KUKA KRL program: EPS_2_25694_BP03_A_20251120043200.src

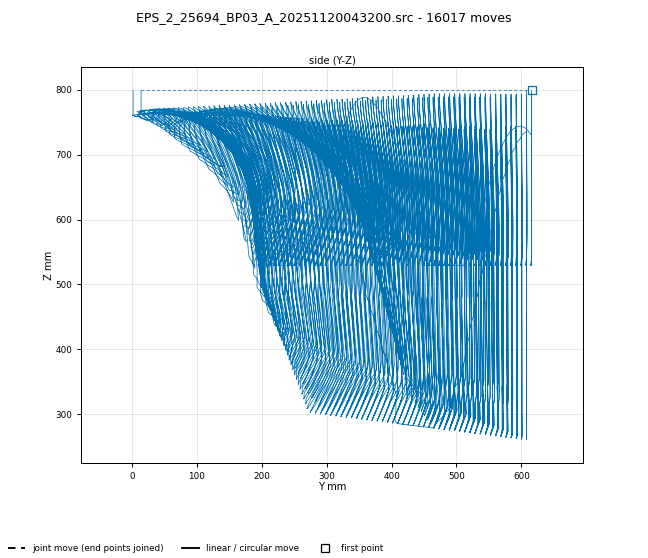
[picture p0: tool path of EPS_2_25694_BP03_A_20251120043200.src, 16017 of 16019 moves have a stored position in this frame; points joined in program order, loops and branches not executed]
&ACCESS RVP
&REL 4
&COMMENT QRS 19112012
&PARAM EDITMASK = *
DEF PART()
EXT BAS (BAS_COMMAND :IN,REAL :IN )
INT I
BAS (#INITMOV,0 )

;KUKA QRS Post kuka4.cps  Date:22-06-2017 !

File_ID=2926

QRS_PRE_INIT()

;Init var - Until changes are made in qrs_pre_init
Outlet_Square_prg=0
Inlet_1_Square_prg=0
Inlet_2_Square_prg=0
Inlet_3_Square_prg=0
Inlet_4_Square_prg=0
Inlet_5_Square_prg=0

Outlet_1={X 0.000, Y 466.000, Z 560.500, B 0.000, E1 0.000 }
Outlet_1={X 0.000, Y 466.000, Z 560.500, B 0.000, E1 0.000 }
Inlet_1={X 0.000, Y 466.000, Z 548.500, B 0.000, E1 90.000 }
Inlet_2={X 0.000, Y 519.840, Z 613.500, B 0.000, E1 205.000 }
Inlet_1={X 0.000, Y 466.000, Z 548.500, B 0.000, E1 90.000 }
Inlet_2={X 0.000, Y 519.840, Z 613.500, B 0.000, E1 205.000 }
Outlet_1_type=457
Inlet_1_type=381
Inlet_2_type=251
Inlet_1_type=381
Inlet_2_type=251
;QRS#1=Sidecore dimensions
;QRS#2=450-18" Concrete
;QRS#3=375-15" Concrete
;QRS#4=250-10" PVC SDR 35
;QRS#5=
;QRS#6=
;QRS#7=
;QRS#8=
;QRS#9=28A PSX-2
;QRS#10=24L PSX-2
;QRS#11=14M PSX
;QRS#12=
;QRS#13=
;QRS#14=
;QRS#15=
;QRS#16=1220x127x1143 3,75'
;QRS#17=EPS Height
;QRS#18=789
;QRS#19=*
;QRS#20= UPDATED VERSION 22-06-2017
;QRS#21=*
Outlet_Square=0250
Inlet_1_Square=0150
Inlet_2_Square=0100
Inlet_3_Square=0
Inlet_4_Square=0
Inlet_5_Square=0
Mill_Square=1
Outlet_Square_Prg=274
Inlet_1_Square_prg=261
Inlet_2_Square_prg=205
Inlet_1_Square_prg=261
Inlet_2_Square_prg=205

QRS_INIT()

$ADVANCE=5

; T1
PTP {E1 172.387,E2 172.387}
PTP {X 0,Y 615.713,A -85,B 0,C 180,E1 172.387,E2 172.387,E3 0,E4 0,E5 0,E6 0}
QRS_SPEED_INIT()
LIN {X 0,Y 615.713,Z 799,A -85,B 0,C 180,E1 172.387,E2 172.387,E3 0,E4 0,E5 0,E6 0} C_VEL
LIN {X 0,Y 615.713,Z 739.037,A -85,B 0,C 180,E1 172.387,E2 172.387} C_VEL
LIN {X 0,Y 615.713,Z 731.107,A -85,B 0,C 180,E1 172.387,E2 172.387} C_VEL
LIN {X 0,Y 615.691,Z 729.212,A -85,B 0,C 180,E1 172.633,E2 172.633} C_VEL
LIN {X 0,Y 615.732,Z 733.219,A -85,B 0,C 180,E1 173.736,E2 173.736} C_VEL
LIN {X 0,Y 615.814,Z 736.045,A -85,B 0,C 180,E1 174.659,E2 174.659} C_VEL
LIN {X 0,Y 615.663,Z 738.454,A -85,B 0,C 180,E1 175.589,E2 175.589} C_VEL
LIN {X 0,Y 615.667,Z 740.356,A -85,B 0,C 180,E1 176.519,E2 176.519} C_VEL
LIN {X 0,Y 615.819,Z 741.763,A -85,B 0,C 180,E1 177.448,E2 177.448} C_VEL
LIN {X 0,Y 615.624,Z 743.112,A -85,B 0,C 180,E1 178.84,E2 178.84} C_VEL
LIN {X 0,Y 615.601,Z 743.434,A -85,B 0,C 180,E1 179.768,E2 179.768} C_VEL
LIN {X 0,Y 615.739,Z 743.277,A -85,B 0,C 180,E1 180.696,E2 180.696} C_VEL
LIN {X 0,Y 615.854,Z 743.003,A -85,B 0,C 180,E1 181.159,E2 181.159} C_VEL
LIN {X 0,Y 615.71,Z 742.227,A -85,B 0,C 180,E1 182.088,E2 182.088} C_VEL
LIN {X 0,Y 615.687,Z 741.683,A -85,B 0,C 180,E1 182.552,E2 182.552} C_VEL
LIN {X 0,Y 615.745,Z 740.192,A -85,B 0,C 180,E1 183.481,E2 183.481} C_VEL
LIN {X 0,Y 615.79,Z 738.236,A -85,B 0,C 180,E1 184.41,E2 184.41} C_VEL
LIN {X 0,Y 615.65,Z 735.834,A -85,B 0,C 180,E1 185.342,E2 185.342} C_VEL
LIN {X 0,Y 615.661,Z 733.002,A -85,B 0,C 180,E1 186.247,E2 186.247} C_VEL
LIN {X 0,Y 615.81,Z 729.772,A -85,B 0,C 180,E1 187.122,E2 187.122} C_VEL
LIN {X 0,Y 615.717,Z 725.49,A -85,B 0,C 180,E1 188.145,E2 188.145} C_VEL
LIN {X 0,Y 615.668,Z 721.228,A -85,B 0,C 180,E1 189.025,E2 189.025} C_VEL
LIN {X 0,Y 615.787,Z 716.395,A -85,B 0,C 180,E1 189.905,E2 189.905} C_VEL
LIN {X 0,Y 615.78,Z 710.979,A -85,B 0,C 180,E1 190.789,E2 190.789} C_VEL
LIN {X 0,Y 615.717,Z 704.917,A -85,B 0,C 180,E1 191.677,E2 191.677} C_VEL
LIN {X 0,Y 615.775,Z 699.333,A -85,B 0,C 180,E1 192.417,E2 192.417} C_VEL
LIN {X 0,Y 615.828,Z 693.198,A -85,B 0,C 180,E1 193.158,E2 193.158} C_VEL
LIN {X 0,Y 615.758,Z 686.46,A -85,B 0,C 180,E1 193.905,E2 193.905} C_VEL
LIN {X 0,Y 615.758,Z 680.597,A -85,B 0,C 180,E1 194.503,E2 194.503} C_VEL
LIN {X 0,Y 615.803,Z 672.516,A -85,B 0,C 180,E1 195.252,E2 195.252} C_VEL
LIN {X 0,Y 615.785,Z 665.226,A -85,B 0,C 180,E1 195.871,E2 195.871} C_VEL
LIN {X 0,Y 615.783,Z 657.531,A -85,B 0,C 180,E1 196.468,E2 196.468} C_VEL
LIN {X 0,Y 615.772,Z 649.053,A -85,B 0,C 180,E1 197.069,E2 197.069} C_VEL
LIN {X 0,Y 615.777,Z 641.285,A -85,B 0,C 180,E1 197.571,E2 197.571} C_VEL
LIN {X 0,Y 615.791,Z 633.21,A -85,B 0,C 180,E1 198.046,E2 198.046} C_VEL
LIN {X 0,Y 615.786,Z 624.289,A -85,B 0,C 180,E1 198.521,E2 198.521} C_VEL
LIN {X 0,Y 615.708,Z 614.895,A -85,B 0,C 180,E1 198.971,E2 198.971} C_VEL
LIN {X 0,Y 615.796,Z 605.823,A -85,B 0,C 180,E1 199.352,E2 199.352} C_VEL
LIN {X 0,Y 615.802,Z 596.522,A -85,B 0,C 180,E1 199.698,E2 199.698} C_VEL
LIN {X 0,Y 615.75,Z 586.286,A -85,B 0,C 180,E1 200.027,E2 200.027} C_VEL
LIN {X 0,Y 615.701,Z 578.595,A -85,B 0,C 180,E1 200.243,E2 200.243} C_VEL
LIN {X 0,Y 615.799,Z 567.336,A -85,B 0,C 180,E1 200.495,E2 200.495} C_VEL
LIN {X 0,Y 615.798,Z 557.38,A -85,B 0,C 180,E1 200.672,E2 200.672} C_VEL
LIN {X 0,Y 615.482,Z 537.657,A -85,B 0,C 180,E1 200.94,E2 200.94} C_VEL
LIN {X 0,Y 615.266,Z 529.66,A -85,B 0,C 180,E1 201.046,E2 201.046} C_VEL
LIN {X 0,Y 615.471,Z 529.66,A -85,B 0,C 180,E1 201.079,E2 201.079} C_VEL
LIN {X 0,Y 615.868,Z 529.66,A -85,B 0,C 180,E1 201.381,E2 201.381} C_VEL
LIN {X 0,Y 615.844,Z 529.66,A -85,B 0,C 180,E1 202.61,E2 202.61} C_VEL
LIN {X 0,Y 615.752,Z 529.66,A -85,B 0,C 180,E1 207.74,E2 207.74} C_VEL
LIN {X 0,Y 615.186,Z 529.66,A -85,B 0,C 180,E1 210.425,E2 210.425} C_VEL
LIN {X 0,Y 615.704,Z 529.66,A -85,B 0,C 180,E1 213.124,E2 213.124} C_VEL
LIN {X 0,Y 615.633,Z 529.66,A -85,B 0,C 180,E1 213.911,E2 213.911} C_VEL
LIN {X 0,Y 615.66,Z 529.66,A -85,B 0,C 180,E1 218.863,E2 218.863} C_VEL
LIN {X 0,Y 615.247,Z 529.66,A -85,B 0,C 180,E1 221.943,E2 221.943} C_VEL
LIN {X 0,Y 615.648,Z 529.66,A -85,B 0,C 180,E1 224.892,E2 224.892} C_VEL
LIN {X 0,Y 615.652,Z 529.66,A -85,B 0,C 180,E1 228.496,E2 228.496} C_VEL
LIN {X 0,Y 615.387,Z 529.66,A -85,B 0,C 180,E1 231.116,E2 231.116} C_VEL
LIN {X 0,Y 615.438,Z 529.66,A -85,B 0,C 180,E1 232.155,E2 232.155} C_VEL
LIN {X 0,Y 615.703,Z 529.66,A -85,B 0,C 180,E1 234.059,E2 234.059} C_VEL
LIN {X 0,Y 615.162,Z 529.66,A -85,B 0,C 180,E1 236.842,E2 236.842} C_VEL
LIN {X 0,Y 615.753,Z 529.66,A -85,B 0,C 180,E1 239.606,E2 239.606} C_VEL
LIN {X 0,Y 615.248,Z 529.66,A -85,B 0,C 180,E1 242.234,E2 242.234} C_VEL
LIN {X 0,Y 615.196,Z 529.66,A -85,B 0,C 180,E1 244.825,E2 244.825} C_VEL
LIN {X 0,Y 614.949,Z 529.66,A -85,B 0,C 180,E1 244.857,E2 244.857} C_VEL
LIN {X 0,Y 615.521,Z 542.401,A -85,B 0,C 180,E1 245.055,E2 245.055} C_VEL
LIN {X 0,Y 615.592,Z 572.277,A -85,B 0,C 180,E1 245.446,E2 245.446} C_VEL
LIN {X 0,Y 615.552,Z 581.408,A -85,B 0,C 180,E1 245.594,E2 245.594} C_VEL
LIN {X 0,Y 615.691,Z 592.991,A -85,B 0,C 180,E1 245.841,E2 245.841} C_VEL
LIN {X 0,Y 615.671,Z 604.649,A -85,B 0,C 180,E1 246.141,E2 246.141} C_VEL
LIN {X 0,Y 615.619,Z 614.365,A -85,B 0,C 180,E1 246.431,E2 246.431} C_VEL
LIN {X 0,Y 615.762,Z 626.855,A -85,B 0,C 180,E1 246.881,E2 246.881} C_VEL
LIN {X 0,Y 615.772,Z 637.702,A -85,B 0,C 180,E1 247.323,E2 247.323} C_VEL
LIN {X 0,Y 615.696,Z 648.639,A -85,B 0,C 180,E1 247.826,E2 247.826} C_VEL
LIN {X 0,Y 615.747,Z 658.322,A -85,B 0,C 180,E1 248.324,E2 248.324} C_VEL
LIN {X 0,Y 615.764,Z 669.199,A -85,B 0,C 180,E1 248.948,E2 248.948} C_VEL
LIN {X 0,Y 615.755,Z 679.009,A -85,B 0,C 180,E1 249.567,E2 249.567} C_VEL
LIN {X 0,Y 615.75,Z 688.977,A -85,B 0,C 180,E1 250.261,E2 250.261} C_VEL
LIN {X 0,Y 615.756,Z 698.046,A -85,B 0,C 180,E1 250.953,E2 250.953} C_VEL
LIN {X 0,Y 615.778,Z 707.426,A -85,B 0,C 180,E1 251.737,E2 251.737} C_VEL
LIN {X 0,Y 615.74,Z 715.07,A -85,B 0,C 180,E1 252.428,E2 252.428} C_VEL
LIN {X 0,Y 615.695,Z 722.27,A -85,B 0,C 180,E1 253.13,E2 253.13} C_VEL
LIN {X 0,Y 615.739,Z 730.247,A -85,B 0,C 180,E1 253.981,E2 253.981} C_VEL
LIN {X 0,Y 615.804,Z 736.878,A -85,B 0,C 180,E1 254.747,E2 254.747} C_VEL
LIN {X 0,Y 615.686,Z 744.025,A -85,B 0,C 180,E1 255.644,E2 255.644} C_VEL
LIN {X 0,Y 615.686,Z 750.525,A -85,B 0,C 180,E1 256.54,E2 256.54} C_VEL
LIN {X 0,Y 615.815,Z 756.425,A -85,B 0,C 180,E1 257.435,E2 257.435} C_VEL
LIN {X 0,Y 615.707,Z 761.804,A -85,B 0,C 180,E1 258.322,E2 258.322} C_VEL
LIN {X 0,Y 615.618,Z 768.146,A -85,B 0,C 180,E1 259.503,E2 259.503} C_VEL
LIN {X 0,Y 615.746,Z 772.394,A -85,B 0,C 180,E1 260.388,E2 260.388} C_VEL
LIN {X 0,Y 615.772,Z 776.164,A -85,B 0,C 180,E1 261.269,E2 261.269} C_VEL
LIN {X 0,Y 615.627,Z 781.078,A -85,B 0,C 180,E1 262.578,E2 262.578} C_VEL
LIN {X 0,Y 615.759,Z 784.681,A -85,B 0,C 180,E1 263.749,E2 263.749} C_VEL
LIN {X 0,Y 615.831,Z 785.856,A -85,B 0,C 180,E1 264.192,E2 264.192} C_VEL
LIN {X 0,Y 615.723,Z 787.098,A -85,B 0,C 180,E1 264.657,E2 264.657} C_VEL
LIN {X 0,Y 615.589,Z 789.148,A -85,B 0,C 180,E1 265.587,E2 265.587} C_VEL
LIN {X 0,Y 615.603,Z 790.751,A -85,B 0,C 180,E1 266.518,E2 266.518} C_VEL
LIN {X 0,Y 615.787,Z 791.942,A -85,B 0,C 180,E1 267.447,E2 267.447} C_VEL
LIN {X 0,Y 615.603,Z 793.162,A -85,B 0,C 180,E1 268.839,E2 268.839} C_VEL
LIN {X 0,Y 615.579,Z 793.427,A -85,B 0,C 180,E1 269.767,E2 269.767} C_VEL
LIN {X 0,Y 615.832,Z 793.119,A -85,B 0,C 180,E1 271.158,E2 271.158} C_VEL
LIN {X 0,Y 615.72,Z 792.484,A -85,B 0,C 180,E1 272.087,E2 272.087} C_VEL
LIN {X 0,Y 615.801,Z 790.717,A -85,B 0,C 180,E1 273.479,E2 273.479} C_VEL
LIN {X 0,Y 615.711,Z 789.131,A -85,B 0,C 180,E1 274.41,E2 274.41} C_VEL
LIN {X 0,Y 615.574,Z 787.129,A -85,B 0,C 180,E1 275.342,E2 275.342} C_VEL
LIN {X 0,Y 615.634,Z 784.612,A -85,B 0,C 180,E1 276.287,E2 276.287} C_VEL
LIN {X 0,Y 615.792,Z 780.631,A -85,B 0,C 180,E1 277.55,E2 277.55} C_VEL
LIN {X 0,Y 615.625,Z 776.195,A -85,B 0,C 180,E1 278.731,E2 278.731} C_VEL
LIN {X 0,Y 615.66,Z 772.414,A -85,B 0,C 180,E1 279.611,E2 279.611} C_VEL
LIN {X 0,Y 615.799,Z 766.633,A -85,B 0,C 180,E1 280.787,E2 280.787} C_VEL
LIN {X 0,Y 615.638,Z 761.823,A -85,B 0,C 180,E1 281.677,E2 281.677} C_VEL
LIN {X 0,Y 615.663,Z 754.512,A -85,B 0,C 180,E1 282.863,E2 282.863} C_VEL
LIN {X 0,Y 615.826,Z 748.416,A -85,B 0,C 180,E1 283.753,E2 283.753} C_VEL
LIN {X 0,Y 615.735,Z 741.72,A -85,B 0,C 180,E1 284.653,E2 284.653} C_VEL
LIN {X 0,Y 615.701,Z 734.344,A -85,B 0,C 180,E1 285.553,E2 285.553} C_VEL
LIN {X 0,Y 615.778,Z 727.648,A -85,B 0,C 180,E1 286.305,E2 286.305} C_VEL
LIN {X 0,Y 615.765,Z 719.307,A -85,B 0,C 180,E1 287.163,E2 287.163} C_VEL
LIN {X 0,Y 615.713,Z 710.778,A -85,B 0,C 180,E1 287.968,E2 287.968} C_VEL
LIN {X 0,Y 615.737,Z 702.667,A -85,B 0,C 180,E1 288.671,E2 288.671} C_VEL
LIN {X 0,Y 615.745,Z 694.151,A -85,B 0,C 180,E1 289.352,E2 289.352} C_VEL
LIN {X 0,Y 615.759,Z 684.699,A -85,B 0,C 180,E1 290.045,E2 290.045} C_VEL
LIN {X 0,Y 615.742,Z 675.485,A -85,B 0,C 180,E1 290.663,E2 290.663} C_VEL
LIN {X 0,Y 615.716,Z 665.295,A -85,B 0,C 180,E1 291.285,E2 291.285} C_VEL
LIN {X 0,Y 615.75,Z 655.432,A -85,B 0,C 180,E1 291.83,E2 291.83} C_VEL
LIN {X 0,Y 615.747,Z 644.949,A -85,B 0,C 180,E1 292.352,E2 292.352} C_VEL
LIN {X 0,Y 615.698,Z 633.849,A -85,B 0,C 180,E1 292.844,E2 292.844} C_VEL
LIN {X 0,Y 615.669,Z 623.571,A -85,B 0,C 180,E1 293.249,E2 293.249} C_VEL
LIN {X 0,Y 615.734,Z 610.394,A -85,B 0,C 180,E1 293.687,E2 293.687} C_VEL
LIN {X 0,Y 615.669,Z 598.849,A -85,B 0,C 180,E1 294.016,E2 294.016} C_VEL
LIN {X 0,Y 615.62,Z 590.562,A -85,B 0,C 180,E1 294.221,E2 294.221} C_VEL
LIN {X 0,Y 615.768,Z 576.553,A -85,B 0,C 180,E1 294.483,E2 294.483} C_VEL
LIN {X 0,Y 615.688,Z 559.539,A -85,B 0,C 180,E1 294.722,E2 294.722} C_VEL
LIN {X 0,Y 615.448,Z 539.088,A -85,B 0,C 180,E1 294.99,E2 294.99} C_VEL
LIN {X 0,Y 614.945,Z 529.66,A -85,B 0,C 180,E1 295.141,E2 295.141} C_VEL
LIN {X 0,Y 615.189,Z 529.66,A -85,B 0,C 180,E1 295.173,E2 295.173} C_VEL
LIN {X 0,Y 615.248,Z 529.66,A -85,B 0,C 180,E1 297.764,E2 297.764} C_VEL
LIN {X 0,Y 615.753,Z 529.66,A -85,B 0,C 180,E1 300.392,E2 300.392} C_VEL
LIN {X 0,Y 615.154,Z 529.66,A -85,B 0,C 180,E1 303.845,E2 303.845} C_VEL
LIN {X 0,Y 615.702,Z 529.66,A -85,B 0,C 180,E1 305.938,E2 305.938} C_VEL
LIN {X 0,Y 615.768,Z 529.66,A -85,B 0,C 180,E1 308.853,E2 308.853} C_VEL
LIN {X 0,Y 615.261,Z 529.66,A -85,B 0,C 180,E1 311.94,E2 311.94} C_VEL
LIN {X 0,Y 615.681,Z 529.66,A -85,B 0,C 180,E1 314.895,E2 314.895} C_VEL
LIN {X 0,Y 615.647,Z 529.66,A -85,B 0,C 180,E1 318.495,E2 318.495} C_VEL
LIN {X 0,Y 615.364,Z 529.66,A -85,B 0,C 180,E1 321.115,E2 321.115} C_VEL
LIN {X 0,Y 615.416,Z 529.66,A -85,B 0,C 180,E1 322.155,E2 322.155} C_VEL
LIN {X 0,Y 615.67,Z 529.66,A -85,B 0,C 180,E1 324.058,E2 324.058} C_VEL
LIN {X 0,Y 615.141,Z 529.66,A -85,B 0,C 180,E1 326.841,E2 326.841} C_VEL
LIN {X 0,Y 615.744,Z 529.66,A -85,B 0,C 180,E1 329.606,E2 329.606} C_VEL
LIN {X 0,Y 615.231,Z 529.66,A -85,B 0,C 180,E1 332.234,E2 332.234} C_VEL
LIN {X 0,Y 615.765,Z 529.66,A -85,B 0,C 180,E1 334.851,E2 334.851} C_VEL
LIN {X 0,Y 615.775,Z 529.66,A -85,B 0,C 180,E1 339.878,E2 339.878} C_VEL
LIN {X 0,Y 615.792,Z 529.66,A -85,B 0,C 180,E1 343.784,E2 343.784} C_VEL
LIN {X 0,Y 615.824,Z 529.66,A -85,B 0,C 180,E1 349.507,E2 349.507} C_VEL
LIN {X 0,Y 615.819,Z 529.66,A -85,B 0,C 180,E1 354.193,E2 354.193} C_VEL
LIN {X 0,Y 615.867,Z 529.66,A -85,B 0,C 180,E1 358.841,E2 358.841} C_VEL
LIN {X 0,Y 615.87,Z 529.66,A -85,B 0,C 180,E1 363.48,E2 363.48} C_VEL
LIN {X 0,Y 615.807,Z 529.66,A -85,B 0,C 180,E1 368.143,E2 368.143} C_VEL
LIN {X 0,Y 615.817,Z 529.66,A -85,B 0,C 180,E1 372.861,E2 372.861} C_VEL
LIN {X 0,Y 615.8,Z 529.66,A -85,B 0,C 180,E1 377.67,E2 377.67} C_VEL
LIN {X 0,Y 615.799,Z 529.66,A -85,B 0,C 180,E1 377.998,E2 377.998} C_VEL
LIN {X 0,Y 615.759,Z 529.66,A -85,B 0,C 180,E1 382.613,E2 382.613} C_VEL
LIN {X 0,Y 615.223,Z 529.66,A -85,B 0,C 180,E1 385.173,E2 385.173} C_VEL
LIN {X 0,Y 615.722,Z 529.66,A -85,B 0,C 180,E1 387.742,E2 387.742} C_VEL
LIN {X 0,Y 615.171,Z 529.66,A -85,B 0,C 180,E1 390.426,E2 390.426} C_VEL
LIN {X 0,Y 615.705,Z 529.66,A -85,B 0,C 180,E1 393.124,E2 393.124} C_VEL
LIN {X 0,Y 615.647,Z 529.66,A -85,B 0,C 180,E1 393.916,E2 393.916} C_VEL
LIN {X 0,Y 615.662,Z 529.66,A -85,B 0,C 180,E1 398.863,E2 398.863} C_VEL
LIN {X 0,Y 615.226,Z 529.66,A -85,B 0,C 180,E1 401.945,E2 401.945} C_VEL
LIN {X 0,Y 615.622,Z 529.66,A -85,B 0,C 180,E1 404.892,E2 404.892} C_VEL
LIN {X 0,Y 615.63,Z 529.66,A -85,B 0,C 180,E1 408.499,E2 408.499} C_VEL
LIN {X 0,Y 615.634,Z 529.66,A -85,B 0,C 180,E1 409.224,E2 409.224} C_VEL
LIN {X 0,Y 614.905,Z 529.66,A -85,B 0,C 180,E1 409.372,E2 409.372} C_VEL
LIN {X 0,Y 614.377,Z 529.66,A -85,B 0,C 180,E1 409.433,E2 409.433} C_VEL
LIN {X 0,Y 614.179,Z 530.164,A -85,B 0,C 180,E1 409.484,E2 409.484} C_VEL
LIN {X 0,Y 615.256,Z 532.913,A -85,B 0,C 180,E1 409.545,E2 409.545} C_VEL
LIN {X 0,Y 615.716,Z 535.143,A -85,B 0,C 180,E1 409.583,E2 409.583} C_VEL
LIN {X 0,Y 615.768,Z 609.489,A -85,B 0,C 180,E1 410.467,E2 410.467} C_VEL
LIN {X 0,Y 615.796,Z 617.276,A -85,B 0,C 180,E1 410.59,E2 410.59} C_VEL
LIN {X 0,Y 615.762,Z 625.824,A -85,B 0,C 180,E1 410.767,E2 410.767} C_VEL
LIN {X 0,Y 615.8,Z 635.584,A -85,B 0,C 180,E1 411.03,E2 411.03} C_VEL
LIN {X 0,Y 615.784,Z 644.692,A -85,B 0,C 180,E1 411.34,E2 411.34} C_VEL
LIN {X 0,Y 615.833,Z 653.267,A -85,B 0,C 180,E1 411.687,E2 411.687} C_VEL
LIN {X 0,Y 615.837,Z 663.366,A -85,B 0,C 180,E1 412.173,E2 412.173} C_VEL
LIN {X 0,Y 615.838,Z 670.383,A -85,B 0,C 180,E1 412.565,E2 412.565} C_VEL
LIN {X 0,Y 615.802,Z 678.254,A -85,B 0,C 180,E1 413.06,E2 413.06} C_VEL
LIN {X 0,Y 615.823,Z 685.634,A -85,B 0,C 180,E1 413.59,E2 413.59} C_VEL
LIN {X 0,Y 615.832,Z 693.033,A -85,B 0,C 180,E1 414.194,E2 414.194} C_VEL
LIN {X 0,Y 615.776,Z 699.754,A -85,B 0,C 180,E1 414.807,E2 414.807} C_VEL
LIN {X 0,Y 615.778,Z 705.651,A -85,B 0,C 180,E1 415.419,E2 415.419} C_VEL
LIN {X 0,Y 615.83,Z 711.178,A -85,B 0,C 180,E1 416.062,E2 416.062} C_VEL
LIN {X 0,Y 615.759,Z 717.457,A -85,B 0,C 180,E1 416.881,E2 416.881} C_VEL
LIN {X 0,Y 615.743,Z 722.895,A -85,B 0,C 180,E1 417.715,E2 417.715} C_VEL
LIN {X 0,Y 615.829,Z 726.982,A -85,B 0,C 180,E1 418.434,E2 418.434} C_VEL
LIN {X 0,Y 615.789,Z 730.525,A -85,B 0,C 180,E1 419.14,E2 419.14} C_VEL
LIN {X 0,Y 615.712,Z 734.28,A -85,B 0,C 180,E1 420.032,E2 420.032} C_VEL
LIN {X 0,Y 615.725,Z 735.961,A -85,B 0,C 180,E1 420.488,E2 420.488} C_VEL
LIN {X 0,Y 615.843,Z 738.595,A -85,B 0,C 180,E1 421.365,E2 421.365} C_VEL
LIN {X 0,Y 615.741,Z 740.746,A -85,B 0,C 180,E1 422.261,E2 422.261} C_VEL
LIN {X 0,Y 615.727,Z 741.895,A -85,B 0,C 180,E1 422.913,E2 422.913} C_VEL
LIN {X 0,Y 615.792,Z 742.709,A -85,B 0,C 180,E1 423.565,E2 423.565} C_VEL
LIN {X 0,Y 615.815,Z 743.213,A -85,B 0,C 180,E1 424.212,E2 424.212} C_VEL
LIN {X 0,Y 615.733,Z 743.429,A -85,B 0,C 180,E1 424.851,E2 424.851} C_VEL
LIN {X 0,Y 615.737,Z 743.29,A -85,B 0,C 180,E1 425.605,E2 425.605} C_VEL
LIN {X 0,Y 615.851,Z 742.529,A -85,B 0,C 180,E1 426.486,E2 426.486} C_VEL
LIN {X 0,Y 615.727,Z 741.246,A -85,B 0,C 180,E1 427.387,E2 427.387} C_VEL
LIN {X 0,Y 615.686,Z 739.971,A -85,B 0,C 180,E1 428.012,E2 428.012} C_VEL
LIN {X 0,Y 615.727,Z 738.372,A -85,B 0,C 180,E1 428.637,E2 428.637} C_VEL
LIN {X 0,Y 615.814,Z 735.406,A -85,B 0,C 180,E1 429.571,E2 429.571} C_VEL
LIN {X 0,Y 615.73,Z 731.754,A -85,B 0,C 180,E1 430.494,E2 430.494} C_VEL
LIN {X 0,Y 615.777,Z 727.849,A -85,B 0,C 180,E1 431.318,E2 431.318} C_VEL
LIN {X 0,Y 615.82,Z 723.223,A -85,B 0,C 180,E1 432.138,E2 432.138} C_VEL
LIN {X 0,Y 615.771,Z 719.45,A -85,B 0,C 180,E1 432.734,E2 432.734} C_VEL
LIN {X 0,Y 615.775,Z 715.176,A -85,B 0,C 180,E1 433.338,E2 433.338} C_VEL
LIN {X 0,Y 615.841,Z 708.758,A -85,B 0,C 180,E1 434.141,E2 434.141} C_VEL
LIN {X 0,Y 615.801,Z 703.223,A -85,B 0,C 180,E1 434.749,E2 434.749} C_VEL
LIN {X 0,Y 615.796,Z 697.131,A -85,B 0,C 180,E1 435.349,E2 435.349} C_VEL
LIN {X 0,Y 615.844,Z 690.323,A -85,B 0,C 180,E1 435.948,E2 435.948} C_VEL
LIN {X 0,Y 615.841,Z 682.573,A -85,B 0,C 180,E1 436.545,E2 436.545} C_VEL
LIN {X 0,Y 615.837,Z 674.946,A -85,B 0,C 180,E1 437.066,E2 437.066} C_VEL
LIN {X 0,Y 615.813,Z 666.212,A -85,B 0,C 180,E1 437.585,E2 437.585} C_VEL
LIN {X 0,Y 615.845,Z 657.471,A -85,B 0,C 180,E1 438.031,E2 438.031} C_VEL
LIN {X 0,Y 615.83,Z 649.113,A -85,B 0,C 180,E1 438.401,E2 438.401} C_VEL
LIN {X 0,Y 615.771,Z 640.154,A -85,B 0,C 180,E1 438.732,E2 438.732} C_VEL
LIN {X 0,Y 615.831,Z 630.951,A -85,B 0,C 180,E1 439.01,E2 439.01} C_VEL
LIN {X 0,Y 615.801,Z 621.089,A -85,B 0,C 180,E1 439.25,E2 439.25} C_VEL
LIN {X 0,Y 615.781,Z 611.462,A -85,B 0,C 180,E1 439.415,E2 439.415} C_VEL
LIN {X 0,Y 615.609,Z 555.605,A -85,B 0,C 180,E1 440.088,E2 440.088} C_VEL
LIN {X 0,Y 615.309,Z 530.18,A -85,B 0,C 180,E1 440.396,E2 440.396} C_VEL
LIN {X 0,Y 615.401,Z 529.66,A -85,B 0,C 180,E1 440.42,E2 440.42} C_VEL
LIN {X 0,Y 615.834,Z 529.66,A -85,B 0,C 180,E1 440.539,E2 440.539} C_VEL
LIN {X 0,Y 615.861,Z 529.66,A -85,B 0,C 180,E1 446.521,E2 446.521} C_VEL
LIN {X 0,Y 615.873,Z 529.66,A -85,B 0,C 180,E1 451.16,E2 451.16} C_VEL
LIN {X 0,Y 615.873,Z 529.66,A -85,B 0,C 180,E1 455.807,E2 455.807} C_VEL
LIN {X 0,Y 615.788,Z 529.66,A -85,B 0,C 180,E1 460.495,E2 460.495} C_VEL
LIN {X 0,Y 615.769,Z 529.66,A -85,B 0,C 180,E1 465.254,E2 465.254} C_VEL
LIN {X 0,Y 615.782,Z 529.66,A -85,B 0,C 180,E1 470.123,E2 470.123} C_VEL
LIN {X 0,Y 615.745,Z 529.66,A -85,B 0,C 180,E1 475.151,E2 475.151} C_VEL
LIN {X 0,Y 615.396,Z 529.66,A -85,B 0,C 180,E1 479.457,E2 479.457} C_VEL
LIN {X 0,Y 615.719,Z 529.66,A -85,B 0,C 180,E1 480.396,E2 480.396} C_VEL
LIN {X 0,Y 615.15,Z 529.66,A -85,B 0,C 180,E1 483.844,E2 483.844} C_VEL
LIN {X 0,Y 615.698,Z 529.66,A -85,B 0,C 180,E1 485.941,E2 485.941} C_VEL
LIN {X 0,Y 615.668,Z 529.66,A -85,B 0,C 180,E1 487.873,E2 487.873} C_VEL
LIN {X 0,Y 615.757,Z 529.66,A -85,B 0,C 180,E1 488.856,E2 488.856} C_VEL
LIN {X 0,Y 615.253,Z 529.66,A -85,B 0,C 180,E1 491.943,E2 491.943} C_VEL
LIN {X 0,Y 615.673,Z 529.66,A -85,B 0,C 180,E1 494.894,E2 494.894} C_VEL
LIN {X 0,Y 615.655,Z 529.66,A -85,B 0,C 180,E1 498.497,E2 498.497} C_VEL
LIN {X 0,Y 615.36,Z 529.66,A -85,B 0,C 180,E1 501.114,E2 501.114} C_VEL
LIN {X 0,Y 615.396,Z 529.66,A -85,B 0,C 180,E1 502.16,E2 502.16} C_VEL
LIN {X 0,Y 615.651,Z 529.66,A -85,B 0,C 180,E1 504.056,E2 504.056} C_VEL
LIN {X 0,Y 615.118,Z 529.66,A -85,B 0,C 180,E1 506.84,E2 506.84} C_VEL
LIN {X 0,Y 615.715,Z 529.66,A -85,B 0,C 180,E1 509.604,E2 509.604} C_VEL
LIN {X 0,Y 615.228,Z 529.66,A -85,B 0,C 180,E1 512.234,E2 512.234} C_VEL
LIN {X 0,Y 615.796,Z 529.66,A -85,B 0,C 180,E1 514.852,E2 514.852} C_VEL
LIN {X 0,Y 615.831,Z 529.66,A -85,B 0,C 180,E1 518.764,E2 518.764} C_VEL
LIN {X 0,Y 615.602,Z 529.66,A -85,B 0,C 180,E1 518.876,E2 518.876} C_VEL
LIN {X 0,Y 615.779,Z 556.304,A -85,B 0,C 180,E1 519.221,E2 519.221} C_VEL
LIN {X 0,Y 615.741,Z 565.587,A -85,B 0,C 180,E1 519.379,E2 519.379} C_VEL
LIN {X 0,Y 615.667,Z 573.153,A -85,B 0,C 180,E1 519.536,E2 519.536} C_VEL
LIN {X 0,Y 615.78,Z 583.294,A -85,B 0,C 180,E1 519.798,E2 519.798} C_VEL
LIN {X 0,Y 615.784,Z 592.324,A -85,B 0,C 180,E1 520.071,E2 520.071} C_VEL
LIN {X 0,Y 615.688,Z 602.19,A -85,B 0,C 180,E1 520.414,E2 520.414} C_VEL
LIN {X 0,Y 615.79,Z 611.709,A -85,B 0,C 180,E1 520.802,E2 520.802} C_VEL
LIN {X 0,Y 615.797,Z 620.728,A -85,B 0,C 180,E1 521.213,E2 521.213} C_VEL
LIN {X 0,Y 615.785,Z 628.975,A -85,B 0,C 180,E1 521.631,E2 521.631} C_VEL
LIN {X 0,Y 615.757,Z 637.944,A -85,B 0,C 180,E1 522.136,E2 522.136} C_VEL
LIN {X 0,Y 615.78,Z 645.951,A -85,B 0,C 180,E1 522.633,E2 522.633} C_VEL
LIN {X 0,Y 615.797,Z 654.793,A -85,B 0,C 180,E1 523.241,E2 523.241} C_VEL
LIN {X 0,Y 615.791,Z 662.806,A -85,B 0,C 180,E1 523.845,E2 523.845} C_VEL
LIN {X 0,Y 615.765,Z 670.118,A -85,B 0,C 180,E1 524.447,E2 524.447} C_VEL
LIN {X 0,Y 615.769,Z 676.821,A -85,B 0,C 180,E1 525.047,E2 525.047} C_VEL
LIN {X 0,Y 615.814,Z 683.003,A -85,B 0,C 180,E1 525.648,E2 525.648} C_VEL
LIN {X 0,Y 615.765,Z 690.046,A -85,B 0,C 180,E1 526.393,E2 526.393} C_VEL
LIN {X 0,Y 615.709,Z 696.458,A -85,B 0,C 180,E1 527.136,E2 527.136} C_VEL
LIN {X 0,Y 615.756,Z 702.296,A -85,B 0,C 180,E1 527.88,E2 527.88} C_VEL
LIN {X 0,Y 615.831,Z 707.614,A -85,B 0,C 180,E1 528.621,E2 528.621} C_VEL
LIN {X 0,Y 615.73,Z 711.581,A -85,B 0,C 180,E1 529.21,E2 529.21} C_VEL
LIN {X 0,Y 615.661,Z 716.922,A -85,B 0,C 180,E1 530.093,E2 530.093} C_VEL
LIN {X 0,Y 615.762,Z 721.658,A -85,B 0,C 180,E1 530.977,E2 530.977} C_VEL
LIN {X 0,Y 615.79,Z 725.868,A -85,B 0,C 180,E1 531.856,E2 531.856} C_VEL
LIN {X 0,Y 615.691,Z 729.212,A -85,B 0,C 180,E1 532.633,E2 532.633} C_VEL
LIN {X 0,Y 611.74,Z 735.059,A -85,B 0,C 180,E1 534.144,E2 534.144} C_VEL
LIN {X 0,Y 607.783,Z 739.278,A -85,B 0,C 180,E1 535.697,E2 535.697} C_VEL
LIN {X 0,Y 607.763,Z 743.464,A -85,B 0,C 180,E1 538.575,E2 538.575} C_VEL
LIN {X 0,Y 607.922,Z 743.404,A -85,B 0,C 180,E1 541.42,E2 541.42} C_VEL
LIN {X 0,Y 607.899,Z 739.162,A -85,B 0,C 180,E1 544.269,E2 544.269} C_VEL
LIN {X 0,Y 607.883,Z 728.493,A -85,B 0,C 180,E1 547.623,E2 547.623} C_VEL
LIN {X 0,Y 607.939,Z 712.456,A -85,B 0,C 180,E1 550.727,E2 550.727} C_VEL
LIN {X 0,Y 608,Z 692.204,A -85,B 0,C 180,E1 553.453,E2 553.453} C_VEL
LIN {X 0,Y 608.082,Z 667.028,A -85,B 0,C 180,E1 555.931,E2 555.931} C_VEL
LIN {X 0,Y 608.185,Z 638.464,A -85,B 0,C 180,E1 557.972,E2 557.972} C_VEL
LIN {X 0,Y 608.294,Z 606.206,A -85,B 0,C 180,E1 559.586,E2 559.586} C_VEL
LIN {X 0,Y 608.364,Z 572.382,A -85,B 0,C 180,E1 560.649,E2 560.649} C_VEL
LIN {X 0,Y 607.906,Z 529.66,A -85,B 0,C 180,E1 561.38,E2 561.38} C_VEL
LIN {X 0,Y 607.695,Z 529.66,A -85,B 0,C 180,E1 568.148,E2 568.148} C_VEL
LIN {X 0,Y 607.809,Z 529.66,A -85,B 0,C 180,E1 573.103,E2 573.103} C_VEL
LIN {X 0,Y 607.507,Z 529.66,A -85,B 0,C 180,E1 579.646,E2 579.646} C_VEL
LIN {X 0,Y 607.506,Z 529.66,A -85,B 0,C 180,E1 585.934,E2 585.934} C_VEL
LIN {X 0,Y 607.452,Z 529.66,A -85,B 0,C 180,E1 590.357,E2 590.357} C_VEL
LIN {X 0,Y 607.433,Z 529.66,A -85,B 0,C 180,E1 595.155,E2 595.155} C_VEL
LIN {X 0,Y 607.601,Z 529.66,A -85,B 0,C 180,E1 600.365,E2 600.365} C_VEL
LIN {X 0,Y 607.26,Z 529.66,A -85,B 0,C 180,E1 604.503,E2 604.503} C_VEL
LIN {X 0,Y 608.436,Z 561.303,A -85,B 0,C 180,E1 604.986,E2 604.986} C_VEL
LIN {X 0,Y 608.473,Z 599.633,A -85,B 0,C 180,E1 605.701,E2 605.701} C_VEL
LIN {X 0,Y 608.446,Z 636.055,A -85,B 0,C 180,E1 606.96,E2 606.96} C_VEL
LIN {X 0,Y 608.25,Z 670.026,A -85,B 0,C 180,E1 608.727,E2 608.727} C_VEL
LIN {X 0,Y 608.111,Z 700.158,A -85,B 0,C 180,E1 610.879,E2 610.879} C_VEL
LIN {X 0,Y 607.968,Z 728.788,A -85,B 0,C 180,E1 613.601,E2 613.601} C_VEL
LIN {X 0,Y 607.882,Z 751.803,A -85,B 0,C 180,E1 616.543,E2 616.543} C_VEL
LIN {X 0,Y 607.8,Z 769.647,A -85,B 0,C 180,E1 619.631,E2 619.631} C_VEL
LIN {X 0,Y 607.768,Z 782.683,A -85,B 0,C 180,E1 622.869,E2 622.869} C_VEL
LIN {X 0,Y 607.71,Z 789.996,A -85,B 0,C 180,E1 625.729,E2 625.729} C_VEL
LIN {X 0,Y 607.739,Z 793.511,A -85,B 0,C 180,E1 628.578,E2 628.578} C_VEL
LIN {X 0,Y 607.908,Z 793.51,A -85,B 0,C 180,E1 631.423,E2 631.423} C_VEL
LIN {X 0,Y 607.73,Z 788.487,A -85,B 0,C 180,E1 634.986,E2 634.986} C_VEL
LIN {X 0,Y 607.83,Z 778.937,A -85,B 0,C 180,E1 638.208,E2 638.208} C_VEL
LIN {X 0,Y 607.838,Z 764.016,A -85,B 0,C 180,E1 641.456,E2 641.456} C_VEL
LIN {X 0,Y 607.963,Z 744.066,A -85,B 0,C 180,E1 644.545,E2 644.545} C_VEL
LIN {X 0,Y 608.05,Z 718.03,A -85,B 0,C 180,E1 647.513,E2 647.513} C_VEL
LIN {X 0,Y 608.194,Z 688.345,A -85,B 0,C 180,E1 650.042,E2 650.042} C_VEL
LIN {X 0,Y 608.316,Z 654.998,A -85,B 0,C 180,E1 652.133,E2 652.133} C_VEL
LIN {X 0,Y 608.392,Z 620.469,A -85,B 0,C 180,E1 653.653,E2 653.653} C_VEL
LIN {X 0,Y 608.477,Z 586.214,A -85,B 0,C 180,E1 654.613,E2 654.613} C_VEL
LIN {X 0,Y 607.58,Z 531.954,A -85,B 0,C 180,E1 655.428,E2 655.428} C_VEL
LIN {X 0,Y 607.239,Z 529.66,A -85,B 0,C 180,E1 655.538,E2 655.538} C_VEL
LIN {X 0,Y 607.647,Z 529.66,A -85,B 0,C 180,E1 659.78,E2 659.78} C_VEL
LIN {X 0,Y 607.71,Z 529.66,A -85,B 0,C 180,E1 666.58,E2 666.58} C_VEL
LIN {X 0,Y 607.339,Z 529.66,A -85,B 0,C 180,E1 672.133,E2 672.133} C_VEL
LIN {X 0,Y 607.666,Z 529.66,A -85,B 0,C 180,E1 678.158,E2 678.158} C_VEL
LIN {X 0,Y 607.629,Z 529.66,A -85,B 0,C 180,E1 683.418,E2 683.418} C_VEL
LIN {X 0,Y 607.566,Z 529.66,A -85,B 0,C 180,E1 690.377,E2 690.377} C_VEL
LIN {X 0,Y 607.799,Z 529.66,A -85,B 0,C 180,E1 695.038,E2 695.038} C_VEL
LIN {X 0,Y 607.569,Z 529.66,A -85,B 0,C 180,E1 701.165,E2 701.165} C_VEL
LIN {X 0,Y 607.264,Z 529.66,A -85,B 0,C 180,E1 705.614,E2 705.614} C_VEL
LIN {X 0,Y 607.746,Z 529.66,A -85,B 0,C 180,E1 709.993,E2 709.993} C_VEL
LIN {X 0,Y 607.881,Z 529.66,A -85,B 0,C 180,E1 714.303,E2 714.303} C_VEL
LIN {X 0,Y 607.588,Z 529.66,A -85,B 0,C 180,E1 720.002,E2 720.002} C_VEL
LIN {X 0,Y 607.67,Z 529.66,A -85,B 0,C 180,E1 724.274,E2 724.274} C_VEL
LIN {X 0,Y 607.764,Z 529.66,A -85,B 0,C 180,E1 728.569,E2 728.569} C_VEL
LIN {X 0,Y 607.888,Z 529.66,A -85,B 0,C 180,E1 732.911,E2 732.911} C_VEL
LIN {X 0,Y 607.594,Z 529.66,A -85,B 0,C 180,E1 738.838,E2 738.838} C_VEL
LIN {X 0,Y 607.579,Z 529.66,A -85,B 0,C 180,E1 743.416,E2 743.416} C_VEL
LIN {X 0,Y 607.658,Z 529.66,A -85,B 0,C 180,E1 748.155,E2 748.155} C_VEL
LIN {X 0,Y 607.808,Z 529.66,A -85,B 0,C 180,E1 753.108,E2 753.108} C_VEL
LIN {X 0,Y 607.482,Z 529.66,A -85,B 0,C 180,E1 759.641,E2 759.641} C_VEL
LIN {X 0,Y 607.495,Z 529.66,A -85,B 0,C 180,E1 765.931,E2 765.931} C_VEL
LIN {X 0,Y 607.177,Z 529.66,A -85,B 0,C 180,E1 769.131,E2 769.131} C_VEL
LIN {X 0,Y 606.592,Z 530.446,A -85,B 0,C 180,E1 769.289,E2 769.289} C_VEL
LIN {X 0,Y 608.098,Z 542.16,A -85,B 0,C 180,E1 769.47,E2 769.47} C_VEL
LIN {X 0,Y 608.144,Z 624.143,A -85,B 0,C 180,E1 770.546,E2 770.546} C_VEL
LIN {X 0,Y 608.124,Z 652.634,A -85,B 0,C 180,E1 771.488,E2 771.488} C_VEL
LIN {X 0,Y 608.039,Z 678.51,A -85,B 0,C 180,E1 772.92,E2 772.92} C_VEL
LIN {X 0,Y 607.96,Z 701.929,A -85,B 0,C 180,E1 774.882,E2 774.882} C_VEL
LIN {X 0,Y 607.914,Z 721.026,A -85,B 0,C 180,E1 777.267,E2 777.267} C_VEL
LIN {X 0,Y 607.858,Z 734.168,A -85,B 0,C 180,E1 779.82,E2 779.82} C_VEL
LIN {X 0,Y 607.917,Z 740.473,A -85,B 0,C 180,E1 781.86,E2 781.86} C_VEL
LIN {X 0,Y 607.925,Z 743.162,A -85,B 0,C 180,E1 783.461,E2 783.461} C_VEL
LIN {X 0,Y 607.861,Z 743.988,A -85,B 0,C 180,E1 785.037,E2 785.037} C_VEL
LIN {X 0,Y 607.866,Z 741.852,A -85,B 0,C 180,E1 787.369,E2 787.369} C_VEL
LIN {X 0,Y 607.924,Z 734.675,A -85,B 0,C 180,E1 789.953,E2 789.953} C_VEL
LIN {X 0,Y 607.958,Z 722.026,A -85,B 0,C 180,E1 792.485,E2 792.485} C_VEL
LIN {X 0,Y 607.989,Z 704.616,A -85,B 0,C 180,E1 794.749,E2 794.749} C_VEL
LIN {X 0,Y 608.055,Z 682.187,A -85,B 0,C 180,E1 796.729,E2 796.729} C_VEL
LIN {X 0,Y 608.143,Z 655.872,A -85,B 0,C 180,E1 798.278,E2 798.278} C_VEL
LIN {X 0,Y 608.174,Z 627.894,A -85,B 0,C 180,E1 799.275,E2 799.275} C_VEL
LIN {X 0,Y 608.067,Z 586.852,A -85,B 0,C 180,E1 799.905,E2 799.905} C_VEL
LIN {X 0,Y 607.797,Z 529.66,A -85,B 0,C 180,E1 800.612,E2 800.612} C_VEL
LIN {X 0,Y 607.737,Z 529.66,A -85,B 0,C 180,E1 807.153,E2 807.153} C_VEL
LIN {X 0,Y 607.866,Z 529.66,A -85,B 0,C 180,E1 811.422,E2 811.422} C_VEL
LIN {X 0,Y 607.663,Z 529.66,A -85,B 0,C 180,E1 816.622,E2 816.622} C_VEL
LIN {X 0,Y 607.559,Z 529.66,A -85,B 0,C 180,E1 821.46,E2 821.46} C_VEL
LIN {X 0,Y 607.629,Z 529.66,A -85,B 0,C 180,E1 825.853,E2 825.853} C_VEL
LIN {X 0,Y 607.785,Z 529.66,A -85,B 0,C 180,E1 830.339,E2 830.339} C_VEL
LIN {X 0,Y 607.782,Z 529.66,A -85,B 0,C 180,E1 834.965,E2 834.965} C_VEL
LIN {X 0,Y 607.605,Z 529.66,A -85,B 0,C 180,E1 839.781,E2 839.781} C_VEL
LIN {X 0,Y 607.731,Z 529.66,A -85,B 0,C 180,E1 846.577,E2 846.577} C_VEL
LIN {X 0,Y 607.338,Z 529.66,A -85,B 0,C 180,E1 851.806,E2 851.806} C_VEL
LIN {X 0,Y 607.499,Z 529.66,A -85,B 0,C 180,E1 856.082,E2 856.082} C_VEL
LIN {X 0,Y 607.414,Z 529.66,A -85,B 0,C 180,E1 860.364,E2 860.364} C_VEL
LIN {X 0,Y 607.386,Z 529.66,A -85,B 0,C 180,E1 865.149,E2 865.149} C_VEL
LIN {X 0,Y 607.554,Z 529.66,A -85,B 0,C 180,E1 870.376,E2 870.376} C_VEL
LIN {X 0,Y 607.839,Z 529.66,A -85,B 0,C 180,E1 875.035,E2 875.035} C_VEL
LIN {X 0,Y 607.876,Z 529.66,A -85,B 0,C 180,E1 878.591,E2 878.591} C_VEL
LIN {X 0,Y 608.277,Z 575.93,A -85,B 0,C 180,E1 879.344,E2 879.344} C_VEL
LIN {X 0,Y 608.263,Z 610.705,A -85,B 0,C 180,E1 880.51,E2 880.51} C_VEL
LIN {X 0,Y 608.17,Z 642.889,A -85,B 0,C 180,E1 882.21,E2 882.21} C_VEL
LIN {X 0,Y 608.047,Z 672.15,A -85,B 0,C 180,E1 884.425,E2 884.425} C_VEL
LIN {X 0,Y 607.904,Z 697.501,A -85,B 0,C 180,E1 887.089,E2 887.089} C_VEL
LIN {X 0,Y 607.809,Z 717.287,A -85,B 0,C 180,E1 889.99,E2 889.99} C_VEL
LIN {X 0,Y 607.812,Z 730.807,A -85,B 0,C 180,E1 892.867,E2 892.867} C_VEL
LIN {X 0,Y 607.783,Z 739.278,A -85,B 0,C 180,E1 895.697,E2 895.697} C_VEL
LIN {X 0,Y 605.253,Z 741.666,A -85,B 0,C 180,E1 896.89,E2 896.89} C_VEL
LIN {X 0,Y 599.93,Z 743.564,A -85,B 0,C 180,E1 898.698,E2 898.698} C_VEL
LIN {X 0,Y 599.824,Z 743.595,A -85,B 0,C 180,E1 898.908,E2 898.908} C_VEL
LIN {X 0,Y 600.018,Z 743.406,A -85,B 0,C 180,E1 901.439,E2 901.439} C_VEL
LIN {X 0,Y 600.013,Z 739.166,A -85,B 0,C 180,E1 904.325,E2 904.325} C_VEL
LIN {X 0,Y 599.998,Z 729.078,A -85,B 0,C 180,E1 907.585,E2 907.585} C_VEL
LIN {X 0,Y 600.078,Z 713.416,A -85,B 0,C 180,E1 910.708,E2 910.708} C_VEL
LIN {X 0,Y 600.21,Z 692.212,A -85,B 0,C 180,E1 913.631,E2 913.631} C_VEL
LIN {X 0,Y 600.371,Z 666.317,A -85,B 0,C 180,E1 916.201,E2 916.201} C_VEL
LIN {X 0,Y 600.603,Z 636.965,A -85,B 0,C 180,E1 918.302,E2 918.302} C_VEL
LIN {X 0,Y 600.828,Z 604.44,A -85,B 0,C 180,E1 919.91,E2 919.91} C_VEL
LIN {X 0,Y 601.015,Z 570.078,A -85,B 0,C 180,E1 920.969,E2 920.969} C_VEL
LIN {X 0,Y 600.071,Z 529.66,A -85,B 0,C 180,E1 921.647,E2 921.647} C_VEL
LIN {X 0,Y 599.674,Z 529.66,A -85,B 0,C 180,E1 928.559,E2 928.559} C_VEL
LIN {X 0,Y 599.672,Z 529.66,A -85,B 0,C 180,E1 933.861,E2 933.861} C_VEL
LIN {X 0,Y 599.616,Z 529.66,A -85,B 0,C 180,E1 938.984,E2 938.984} C_VEL
LIN {X 0,Y 599.521,Z 529.66,A -85,B 0,C 180,E1 945.191,E2 945.191} C_VEL
LIN {X 0,Y 599.564,Z 529.66,A -85,B 0,C 180,E1 951.009,E2 951.009} C_VEL
LIN {X 0,Y 599.586,Z 529.66,A -85,B 0,C 180,E1 954.631,E2 954.631} C_VEL
LIN {X 0,Y 599.649,Z 529.66,A -85,B 0,C 180,E1 959.783,E2 959.783} C_VEL
LIN {X 0,Y 599.361,Z 530.335,A -85,B 0,C 180,E1 964.177,E2 964.177} C_VEL
LIN {X 0,Y 601.16,Z 542.036,A -85,B 0,C 180,E1 964.412,E2 964.412} C_VEL
LIN {X 0,Y 601.266,Z 591.764,A -85,B 0,C 180,E1 965.192,E2 965.192} C_VEL
LIN {X 0,Y 601.101,Z 627.74,A -85,B 0,C 180,E1 966.319,E2 966.319} C_VEL
LIN {X 0,Y 600.836,Z 661.637,A -85,B 0,C 180,E1 967.949,E2 967.949} C_VEL
LIN {X 0,Y 600.566,Z 694.567,A -85,B 0,C 180,E1 970.17,E2 970.17} C_VEL
LIN {X 0,Y 600.251,Z 723.313,A -85,B 0,C 180,E1 972.794,E2 972.794} C_VEL
LIN {X 0,Y 600.059,Z 747.995,A -85,B 0,C 180,E1 975.808,E2 975.808} C_VEL
LIN {X 0,Y 599.933,Z 766.926,A -85,B 0,C 180,E1 978.938,E2 978.938} C_VEL
LIN {X 0,Y 599.875,Z 781.541,A -85,B 0,C 180,E1 982.412,E2 982.412} C_VEL
LIN {X 0,Y 599.826,Z 789.995,A -85,B 0,C 180,E1 985.672,E2 985.672} C_VEL
LIN {X 0,Y 599.839,Z 793.511,A -85,B 0,C 180,E1 988.559,E2 988.559} C_VEL
LIN {X 0,Y 600.005,Z 793.51,A -85,B 0,C 180,E1 991.442,E2 991.442} C_VEL
LIN {X 0,Y 599.955,Z 789.993,A -85,B 0,C 180,E1 994.328,E2 994.328} C_VEL
LIN {X 0,Y 599.983,Z 780.272,A -85,B 0,C 180,E1 997.952,E2 997.952} C_VEL
LIN {X 0,Y 600.007,Z 765.92,A -85,B 0,C 180,E1 1001.25,E2 1001.25} C_VEL
LIN {X 0,Y 600.154,Z 746.654,A -85,B 0,C 180,E1 1004.377,E2 1004.377} C_VEL
LIN {X 0,Y 600.328,Z 721.12,A -85,B 0,C 180,E1 1007.439,E2 1007.439} C_VEL
LIN {X 0,Y 600.587,Z 691.734,A -85,B 0,C 180,E1 1010.047,E2 1010.047} C_VEL
LIN {X 0,Y 600.855,Z 658.768,A -85,B 0,C 180,E1 1012.216,E2 1012.216} C_VEL
LIN {X 0,Y 601.1,Z 622.674,A -85,B 0,C 180,E1 1013.879,E2 1013.879} C_VEL
LIN {X 0,Y 601.277,Z 587.128,A -85,B 0,C 180,E1 1014.909,E2 1014.909} C_VEL
LIN {X 0,Y 600.379,Z 533.585,A -85,B 0,C 180,E1 1015.734,E2 1015.734} C_VEL
LIN {X 0,Y 599.299,Z 529.66,A -85,B 0,C 180,E1 1015.93,E2 1015.93} C_VEL
LIN {X 0,Y 599.544,Z 529.66,A -85,B 0,C 180,E1 1021.163,E2 1021.163} C_VEL
LIN {X 0,Y 599.759,Z 529.66,A -85,B 0,C 180,E1 1027.146,E2 1027.146} C_VEL
LIN {X 0,Y 599.433,Z 529.66,A -85,B 0,C 180,E1 1033.114,E2 1033.114} C_VEL
LIN {X 0,Y 599.589,Z 529.66,A -85,B 0,C 180,E1 1039.027,E2 1039.027} C_VEL
LIN {X 0,Y 599.555,Z 529.66,A -85,B 0,C 180,E1 1044.631,E2 1044.631} C_VEL
LIN {X 0,Y 599.629,Z 529.66,A -85,B 0,C 180,E1 1049.784,E2 1049.784} C_VEL
LIN {X 0,Y 599.863,Z 529.66,A -85,B 0,C 180,E1 1054.906,E2 1054.906} C_VEL
LIN {X 0,Y 599.722,Z 529.66,A -85,B 0,C 180,E1 1060.909,E2 1060.909} C_VEL
LIN {X 0,Y 599.399,Z 529.66,A -85,B 0,C 180,E1 1065.421,E2 1065.421} C_VEL
LIN {X 0,Y 599.806,Z 529.66,A -85,B 0,C 180,E1 1069.859,E2 1069.859} C_VEL
LIN {X 0,Y 599.981,Z 529.66,A -85,B 0,C 180,E1 1074.228,E2 1074.228} C_VEL
LIN {X 0,Y 599.688,Z 529.66,A -85,B 0,C 180,E1 1080.002,E2 1080.002} C_VEL
LIN {X 0,Y 599.752,Z 529.66,A -85,B 0,C 180,E1 1084.331,E2 1084.331} C_VEL
LIN {X 0,Y 599.818,Z 529.66,A -85,B 0,C 180,E1 1088.684,E2 1088.684} C_VEL
LIN {X 0,Y 599.914,Z 529.66,A -85,B 0,C 180,E1 1093.086,E2 1093.086} C_VEL
LIN {X 0,Y 599.655,Z 529.66,A -85,B 0,C 180,E1 1099.097,E2 1099.097} C_VEL
LIN {X 0,Y 599.586,Z 529.66,A -85,B 0,C 180,E1 1103.747,E2 1103.747} C_VEL
LIN {X 0,Y 599.624,Z 529.66,A -85,B 0,C 180,E1 1108.566,E2 1108.566} C_VEL
LIN {X 0,Y 599.682,Z 529.66,A -85,B 0,C 180,E1 1113.861,E2 1113.861} C_VEL
LIN {X 0,Y 599.603,Z 529.66,A -85,B 0,C 180,E1 1118.99,E2 1118.99} C_VEL
LIN {X 0,Y 599.502,Z 529.66,A -85,B 0,C 180,E1 1125.187,E2 1125.187} C_VEL
LIN {X 0,Y 599.149,Z 529.66,A -85,B 0,C 180,E1 1129.043,E2 1129.043} C_VEL
LIN {X 0,Y 600.515,Z 545.59,A -85,B 0,C 180,E1 1129.311,E2 1129.311} C_VEL
LIN {X 0,Y 600.498,Z 623.915,A -85,B 0,C 180,E1 1130.353,E2 1130.353} C_VEL
LIN {X 0,Y 600.415,Z 653.063,A -85,B 0,C 180,E1 1131.33,E2 1131.33} C_VEL
LIN {X 0,Y 600.281,Z 678.932,A -85,B 0,C 180,E1 1132.791,E2 1132.791} C_VEL
LIN {X 0,Y 600.121,Z 701.136,A -85,B 0,C 180,E1 1134.666,E2 1134.666} C_VEL
LIN {X 0,Y 600.04,Z 719.401,A -85,B 0,C 180,E1 1136.919,E2 1136.919} C_VEL
LIN {X 0,Y 599.994,Z 733.309,A -85,B 0,C 180,E1 1139.541,E2 1139.541} C_VEL
LIN {X 0,Y 599.972,Z 741.631,A -85,B 0,C 180,E1 1142.375,E2 1142.375} C_VEL
LIN {X 0,Y 599.949,Z 743.992,A -85,B 0,C 180,E1 1144.89,E2 1144.89} C_VEL
LIN {X 0,Y 599.989,Z 742.276,A -85,B 0,C 180,E1 1147.142,E2 1147.142} C_VEL
LIN {X 0,Y 600.055,Z 735.222,A -85,B 0,C 180,E1 1149.869,E2 1149.869} C_VEL
LIN {X 0,Y 600.083,Z 722.912,A -85,B 0,C 180,E1 1152.436,E2 1152.436} C_VEL
LIN {X 0,Y 600.141,Z 704.617,A -85,B 0,C 180,E1 1154.878,E2 1154.878} C_VEL
LIN {X 0,Y 600.284,Z 681.644,A -85,B 0,C 180,E1 1156.923,E2 1156.923} C_VEL
LIN {X 0,Y 600.444,Z 655.771,A -85,B 0,C 180,E1 1158.457,E2 1158.457} C_VEL
LIN {X 0,Y 600.519,Z 627.923,A -85,B 0,C 180,E1 1159.46,E2 1159.46} C_VEL
LIN {X 0,Y 600.435,Z 587.208,A -85,B 0,C 180,E1 1160.096,E2 1160.096} C_VEL
LIN {X 0,Y 599.873,Z 529.66,A -85,B 0,C 180,E1 1160.863,E2 1160.863} C_VEL
LIN {X 0,Y 599.843,Z 529.66,A -85,B 0,C 180,E1 1167.115,E2 1167.115} C_VEL
LIN {X 0,Y 599.955,Z 529.66,A -85,B 0,C 180,E1 1171.441,E2 1171.441} C_VEL
LIN {X 0,Y 600.038,Z 529.66,A -85,B 0,C 180,E1 1175.773,E2 1175.773} C_VEL
LIN {X 0,Y 599.62,Z 529.66,A -85,B 0,C 180,E1 1181.614,E2 1181.614} C_VEL
LIN {X 0,Y 599.478,Z 529.66,A -85,B 0,C 180,E1 1186.952,E2 1186.952} C_VEL
LIN {X 0,Y 599.555,Z 529.66,A -85,B 0,C 180,E1 1191.368,E2 1191.368} C_VEL
LIN {X 0,Y 599.773,Z 529.66,A -85,B 0,C 180,E1 1195.322,E2 1195.322} C_VEL
LIN {X 0,Y 599.515,Z 529.66,A -85,B 0,C 180,E1 1201.151,E2 1201.151} C_VEL
LIN {X 0,Y 599.809,Z 529.66,A -85,B 0,C 180,E1 1207.141,E2 1207.141} C_VEL
LIN {X 0,Y 599.441,Z 529.66,A -85,B 0,C 180,E1 1213.109,E2 1213.109} C_VEL
LIN {X 0,Y 599.597,Z 529.66,A -85,B 0,C 180,E1 1219.025,E2 1219.025} C_VEL
LIN {X 0,Y 599.522,Z 529.66,A -85,B 0,C 180,E1 1224.624,E2 1224.624} C_VEL
LIN {X 0,Y 599.607,Z 529.66,A -85,B 0,C 180,E1 1229.778,E2 1229.778} C_VEL
LIN {X 0,Y 599.898,Z 529.66,A -85,B 0,C 180,E1 1234.896,E2 1234.896} C_VEL
LIN {X 0,Y 599.889,Z 529.66,A -85,B 0,C 180,E1 1238.284,E2 1238.284} C_VEL
LIN {X 0,Y 601.014,Z 544.793,A -85,B 0,C 180,E1 1238.53,E2 1238.53} C_VEL
LIN {X 0,Y 600.947,Z 581.424,A -85,B 0,C 180,E1 1239.222,E2 1239.222} C_VEL
LIN {X 0,Y 600.772,Z 615.139,A -85,B 0,C 180,E1 1240.458,E2 1240.458} C_VEL
LIN {X 0,Y 600.511,Z 647.133,A -85,B 0,C 180,E1 1242.259,E2 1242.259} C_VEL
LIN {X 0,Y 600.276,Z 675.33,A -85,B 0,C 180,E1 1244.507,E2 1244.507} C_VEL
LIN {X 0,Y 600.097,Z 698.961,A -85,B 0,C 180,E1 1247.103,E2 1247.103} C_VEL
LIN {X 0,Y 599.945,Z 717.281,A -85,B 0,C 180,E1 1249.858,E2 1249.858} C_VEL
LIN {X 0,Y 599.923,Z 730.806,A -85,B 0,C 180,E1 1252.773,E2 1252.773} C_VEL
LIN {X 0,Y 599.915,Z 739.391,A -85,B 0,C 180,E1 1255.691,E2 1255.691} C_VEL
LIN {X 0,Y 599.863,Z 743.466,A -85,B 0,C 180,E1 1258.557,E2 1258.557} C_VEL
LIN {X 0,Y 599.824,Z 743.595,A -85,B 0,C 180,E1 1258.908,E2 1258.908} C_VEL
LIN {X 0,Y 598.564,Z 743.956,A -85,B 0,C 180,E1 1259.733,E2 1259.733} C_VEL
LIN {X 0,Y 592.059,Z 742.872,A -85,B 0,C 180,E1 1262.08,E2 1262.08} C_VEL
LIN {X 0,Y 592.032,Z 742.632,A -85,B 0,C 180,E1 1262.186,E2 1262.186} C_VEL
LIN {X 0,Y 592.017,Z 737.425,A -85,B 0,C 180,E1 1265.116,E2 1265.116} C_VEL
LIN {X 0,Y 592.095,Z 726.018,A -85,B 0,C 180,E1 1268.425,E2 1268.425} C_VEL
LIN {X 0,Y 592.226,Z 708.763,A -85,B 0,C 180,E1 1271.596,E2 1271.596} C_VEL
LIN {X 0,Y 592.446,Z 686.928,A -85,B 0,C 180,E1 1274.419,E2 1274.419} C_VEL
LIN {X 0,Y 592.734,Z 660.151,A -85,B 0,C 180,E1 1276.929,E2 1276.929} C_VEL
LIN {X 0,Y 593.085,Z 630.391,A -85,B 0,C 180,E1 1278.927,E2 1278.927} C_VEL
LIN {X 0,Y 593.43,Z 597.468,A -85,B 0,C 180,E1 1280.442,E2 1280.442} C_VEL
LIN {X 0,Y 593.669,Z 564.686,A -85,B 0,C 180,E1 1281.351,E2 1281.351} C_VEL
LIN {X 0,Y 592.469,Z 531.883,A -85,B 0,C 180,E1 1281.87,E2 1281.87} C_VEL
LIN {X 0,Y 592.119,Z 529.66,A -85,B 0,C 180,E1 1281.957,E2 1281.957} C_VEL
LIN {X 0,Y 591.733,Z 529.66,A -85,B 0,C 180,E1 1287.321,E2 1287.321} C_VEL
LIN {X 0,Y 591.721,Z 529.66,A -85,B 0,C 180,E1 1294.125,E2 1294.125} C_VEL
LIN {X 0,Y 591.531,Z 529.66,A -85,B 0,C 180,E1 1300.068,E2 1300.068} C_VEL
LIN {X 0,Y 591.586,Z 529.66,A -85,B 0,C 180,E1 1305.575,E2 1305.575} C_VEL
LIN {X 0,Y 591.604,Z 529.66,A -85,B 0,C 180,E1 1310.383,E2 1310.383} C_VEL
LIN {X 0,Y 591.505,Z 529.66,A -85,B 0,C 180,E1 1315.859,E2 1315.859} C_VEL
LIN {X 0,Y 591.587,Z 529.66,A -85,B 0,C 180,E1 1321.012,E2 1321.012} C_VEL
LIN {X 0,Y 591.378,Z 529.66,A -85,B 0,C 180,E1 1323.776,E2 1323.776} C_VEL
LIN {X 0,Y 593.943,Z 540.169,A -85,B 0,C 180,E1 1324.054,E2 1324.054} C_VEL
LIN {X 0,Y 594.084,Z 591.938,A -85,B 0,C 180,E1 1324.876,E2 1324.876} C_VEL
LIN {X 0,Y 593.787,Z 627.742,A -85,B 0,C 180,E1 1326.009,E2 1326.009} C_VEL
LIN {X 0,Y 593.407,Z 662.206,A -85,B 0,C 180,E1 1327.692,E2 1327.692} C_VEL
LIN {X 0,Y 592.979,Z 694.503,A -85,B 0,C 180,E1 1329.9,E2 1329.9} C_VEL
LIN {X 0,Y 592.567,Z 723.313,A -85,B 0,C 180,E1 1332.564,E2 1332.564} C_VEL
LIN {X 0,Y 592.265,Z 748.037,A -85,B 0,C 180,E1 1335.623,E2 1335.623} C_VEL
LIN {X 0,Y 592.078,Z 768.104,A -85,B 0,C 180,E1 1339.023,E2 1339.023} C_VEL
LIN {X 0,Y 591.992,Z 781.541,A -85,B 0,C 180,E1 1342.31,E2 1342.31} C_VEL
LIN {X 0,Y 591.929,Z 789.995,A -85,B 0,C 180,E1 1345.614,E2 1345.614} C_VEL
LIN {X 0,Y 591.939,Z 793.511,A -85,B 0,C 180,E1 1348.54,E2 1348.54} C_VEL
LIN {X 0,Y 592.102,Z 793.511,A -85,B 0,C 180,E1 1351.461,E2 1351.461} C_VEL
LIN {X 0,Y 592.042,Z 789.993,A -85,B 0,C 180,E1 1354.386,E2 1354.386} C_VEL
LIN {X 0,Y 592.095,Z 780.272,A -85,B 0,C 180,E1 1358.058,E2 1358.058} C_VEL
LIN {X 0,Y 592.142,Z 765.921,A -85,B 0,C 180,E1 1361.401,E2 1361.401} C_VEL
LIN {X 0,Y 592.338,Z 746.933,A -85,B 0,C 180,E1 1364.532,E2 1364.532} C_VEL
LIN {X 0,Y 592.635,Z 721.566,A -85,B 0,C 180,E1 1367.625,E2 1367.625} C_VEL
LIN {X 0,Y 593.031,Z 692.316,A -85,B 0,C 180,E1 1370.268,E2 1370.268} C_VEL
LIN {X 0,Y 593.413,Z 660.241,A -85,B 0,C 180,E1 1372.423,E2 1372.423} C_VEL
LIN {X 0,Y 593.809,Z 624.517,A -85,B 0,C 180,E1 1374.123,E2 1374.123} C_VEL
LIN {X 0,Y 594.118,Z 588.187,A -85,B 0,C 180,E1 1375.208,E2 1375.208} C_VEL
LIN {X 0,Y 593.308,Z 535.912,A -85,B 0,C 180,E1 1376.032,E2 1376.032} C_VEL
LIN {X 0,Y 591.389,Z 529.66,A -85,B 0,C 180,E1 1376.225,E2 1376.225} C_VEL
LIN {X 0,Y 591.676,Z 529.66,A -85,B 0,C 180,E1 1380.669,E2 1380.669} C_VEL
LIN {X 0,Y 591.758,Z 529.66,A -85,B 0,C 180,E1 1385.91,E2 1385.91} C_VEL
LIN {X 0,Y 591.488,Z 529.66,A -85,B 0,C 180,E1 1391.553,E2 1391.553} C_VEL
LIN {X 0,Y 591.629,Z 529.66,A -85,B 0,C 180,E1 1396.48,E2 1396.48} C_VEL
LIN {X 0,Y 591.685,Z 529.66,A -85,B 0,C 180,E1 1402.263,E2 1402.263} C_VEL
LIN {X 0,Y 591.476,Z 529.66,A -85,B 0,C 180,E1 1407.607,E2 1407.607} C_VEL
LIN {X 0,Y 591.589,Z 529.66,A -85,B 0,C 180,E1 1412.671,E2 1412.671} C_VEL
LIN {X 0,Y 591.509,Z 529.66,A -85,B 0,C 180,E1 1417.504,E2 1417.504} C_VEL
LIN {X 0,Y 591.769,Z 529.66,A -85,B 0,C 180,E1 1422.184,E2 1422.184} C_VEL
LIN {X 0,Y 591.61,Z 529.66,A -85,B 0,C 180,E1 1428.228,E2 1428.228} C_VEL
LIN {X 0,Y 592.046,Z 529.66,A -85,B 0,C 180,E1 1434.151,E2 1434.151} C_VEL
LIN {X 0,Y 591.787,Z 529.66,A -85,B 0,C 180,E1 1440.002,E2 1440.002} C_VEL
LIN {X 0,Y 591.835,Z 529.66,A -85,B 0,C 180,E1 1444.389,E2 1444.389} C_VEL
LIN {X 0,Y 591.876,Z 529.66,A -85,B 0,C 180,E1 1448.801,E2 1448.801} C_VEL
LIN {X 0,Y 591.682,Z 529.66,A -85,B 0,C 180,E1 1454.271,E2 1454.271} C_VEL
LIN {X 0,Y 591.71,Z 529.66,A -85,B 0,C 180,E1 1459.363,E2 1459.363} C_VEL
LIN {X 0,Y 591.621,Z 529.66,A -85,B 0,C 180,E1 1464.087,E2 1464.087} C_VEL
LIN {X 0,Y 591.604,Z 529.66,A -85,B 0,C 180,E1 1468.99,E2 1468.99} C_VEL
LIN {X 0,Y 591.73,Z 529.66,A -85,B 0,C 180,E1 1474.129,E2 1474.129} C_VEL
LIN {X 0,Y 591.518,Z 529.66,A -85,B 0,C 180,E1 1480.064,E2 1480.064} C_VEL
LIN {X 0,Y 591.561,Z 529.66,A -85,B 0,C 180,E1 1485.583,E2 1485.583} C_VEL
LIN {X 0,Y 591.478,Z 529.66,A -85,B 0,C 180,E1 1488.863,E2 1488.863} C_VEL
LIN {X 0,Y 592.899,Z 551.293,A -85,B 0,C 180,E1 1489.175,E2 1489.175} C_VEL
LIN {X 0,Y 592.854,Z 624.519,A -85,B 0,C 180,E1 1490.174,E2 1490.174} C_VEL
LIN {X 0,Y 592.735,Z 652.682,A -85,B 0,C 180,E1 1491.133,E2 1491.133} C_VEL
LIN {X 0,Y 592.528,Z 678.616,A -85,B 0,C 180,E1 1492.607,E2 1492.607} C_VEL
LIN {X 0,Y 592.305,Z 701.945,A -85,B 0,C 180,E1 1494.614,E2 1494.614} C_VEL
LIN {X 0,Y 592.17,Z 720.33,A -85,B 0,C 180,E1 1496.954,E2 1496.954} C_VEL
LIN {X 0,Y 592.137,Z 732.843,A -85,B 0,C 180,E1 1499.357,E2 1499.357} C_VEL
LIN {X 0,Y 592.119,Z 740.956,A -85,B 0,C 180,E1 1502.007,E2 1502.007} C_VEL
LIN {X 0,Y 592.025,Z 743.86,A -85,B 0,C 180,E1 1504.322,E2 1504.322} C_VEL
LIN {X 0,Y 592.087,Z 743.075,A -85,B 0,C 180,E1 1506.566,E2 1506.566} C_VEL
LIN {X 0,Y 592.14,Z 736.784,A -85,B 0,C 180,E1 1509.483,E2 1509.483} C_VEL
LIN {X 0,Y 592.213,Z 724.911,A -85,B 0,C 180,E1 1512.195,E2 1512.195} C_VEL
LIN {X 0,Y 592.295,Z 707.569,A -85,B 0,C 180,E1 1514.673,E2 1514.673} C_VEL
LIN {X 0,Y 592.494,Z 686.031,A -85,B 0,C 180,E1 1516.748,E2 1516.748} C_VEL
LIN {X 0,Y 592.69,Z 660.372,A -85,B 0,C 180,E1 1518.407,E2 1518.407} C_VEL
LIN {X 0,Y 592.836,Z 632.114,A -85,B 0,C 180,E1 1519.535,E2 1519.535} C_VEL
LIN {X 0,Y 592.875,Z 602.378,A -85,B 0,C 180,E1 1520.107,E2 1520.107} C_VEL
LIN {X 0,Y 591.888,Z 529.66,A -85,B 0,C 180,E1 1521.062,E2 1521.062} C_VEL
LIN {X 0,Y 591.932,Z 529.66,A -85,B 0,C 180,E1 1527.077,E2 1527.077} C_VEL
LIN {X 0,Y 592.045,Z 529.66,A -85,B 0,C 180,E1 1531.46,E2 1531.46} C_VEL
LIN {X 0,Y 591.979,Z 529.66,A -85,B 0,C 180,E1 1536.198,E2 1536.198} C_VEL
LIN {X 0,Y 591.685,Z 529.66,A -85,B 0,C 180,E1 1541.772,E2 1541.772} C_VEL
LIN {X 0,Y 591.722,Z 529.66,A -85,B 0,C 180,E1 1546.291,E2 1546.291} C_VEL
LIN {X 0,Y 591.787,Z 529.66,A -85,B 0,C 180,E1 1550.914,E2 1550.914} C_VEL
LIN {X 0,Y 591.523,Z 529.66,A -85,B 0,C 180,E1 1556.762,E2 1556.762} C_VEL
LIN {X 0,Y 591.643,Z 529.66,A -85,B 0,C 180,E1 1560.67,E2 1560.67} C_VEL
LIN {X 0,Y 591.774,Z 529.66,A -85,B 0,C 180,E1 1565.907,E2 1565.907} C_VEL
LIN {X 0,Y 591.606,Z 529.66,A -85,B 0,C 180,E1 1570.073,E2 1570.073} C_VEL
LIN {X 0,Y 591.605,Z 529.66,A -85,B 0,C 180,E1 1575.576,E2 1575.576} C_VEL
LIN {X 0,Y 591.572,Z 529.66,A -85,B 0,C 180,E1 1580.377,E2 1580.377} C_VEL
LIN {X 0,Y 591.439,Z 529.66,A -85,B 0,C 180,E1 1585.852,E2 1585.852} C_VEL
LIN {X 0,Y 591.562,Z 529.66,A -85,B 0,C 180,E1 1591.008,E2 1591.008} C_VEL
LIN {X 0,Y 591.786,Z 529.66,A -85,B 0,C 180,E1 1596.628,E2 1596.628} C_VEL
LIN {X 0,Y 591.955,Z 529.66,A -85,B 0,C 180,E1 1597.969,E2 1597.969} C_VEL
LIN {X 0,Y 593.602,Z 538.823,A -85,B 0,C 180,E1 1598.173,E2 1598.173} C_VEL
LIN {X 0,Y 593.497,Z 577.648,A -85,B 0,C 180,E1 1598.848,E2 1598.848} C_VEL
LIN {X 0,Y 593.273,Z 611.028,A -85,B 0,C 180,E1 1600.013,E2 1600.013} C_VEL
LIN {X 0,Y 592.929,Z 642.88,A -85,B 0,C 180,E1 1601.737,E2 1601.737} C_VEL
LIN {X 0,Y 592.582,Z 672.231,A -85,B 0,C 180,E1 1604.016,E2 1604.016} C_VEL
LIN {X 0,Y 592.307,Z 697.498,A -85,B 0,C 180,E1 1606.743,E2 1606.743} C_VEL
LIN {X 0,Y 592.115,Z 717.275,A -85,B 0,C 180,E1 1609.722,E2 1609.722} C_VEL
LIN {X 0,Y 592.065,Z 731.915,A -85,B 0,C 180,E1 1612.984,E2 1612.984} C_VEL
LIN {X 0,Y 592.032,Z 740.803,A -85,B 0,C 180,E1 1616.345,E2 1616.345} C_VEL
LIN {X 0,Y 591.946,Z 743.997,A -85,B 0,C 180,E1 1619.998,E2 1619.998} C_VEL
LIN {X 0,Y 592.032,Z 742.632,A -85,B 0,C 180,E1 1622.186,E2 1622.186} C_VEL
LIN {X 0,Y 590.762,Z 741.699,A -85,B 0,C 180,E1 1623.019,E2 1623.019} C_VEL
LIN {X 0,Y 584.232,Z 737.233,A -85,B 0,C 180,E1 1625.262,E2 1625.262} C_VEL
LIN {X 0,Y 584.142,Z 736.694,A -85,B 0,C 180,E1 1625.472,E2 1625.472} C_VEL
LIN {X 0,Y 584.212,Z 726.02,A -85,B 0,C 180,E1 1628.539,E2 1628.539} C_VEL
LIN {X 0,Y 584.383,Z 709.246,A -85,B 0,C 180,E1 1631.679,E2 1631.679} C_VEL
LIN {X 0,Y 584.684,Z 686.932,A -85,B 0,C 180,E1 1634.614,E2 1634.614} C_VEL
LIN {X 0,Y 585.056,Z 660.893,A -85,B 0,C 180,E1 1637.098,E2 1637.098} C_VEL
LIN {X 0,Y 585.527,Z 630.408,A -85,B 0,C 180,E1 1639.181,E2 1639.181} C_VEL
LIN {X 0,Y 585.993,Z 597.658,A -85,B 0,C 180,E1 1640.707,E2 1640.707} C_VEL
LIN {X 0,Y 586.317,Z 563.746,A -85,B 0,C 180,E1 1641.652,E2 1641.652} C_VEL
LIN {X 0,Y 585.374,Z 534.229,A -85,B 0,C 180,E1 1642.119,E2 1642.119} C_VEL
LIN {X 0,Y 584.151,Z 529.66,A -85,B 0,C 180,E1 1642.233,E2 1642.233} C_VEL
LIN {X 0,Y 583.722,Z 529.66,A -85,B 0,C 180,E1 1648.487,E2 1648.487} C_VEL
LIN {X 0,Y 583.722,Z 529.66,A -85,B 0,C 180,E1 1654.659,E2 1654.659} C_VEL
LIN {X 0,Y 583.597,Z 529.66,A -85,B 0,C 180,E1 1660.269,E2 1660.269} C_VEL
LIN {X 0,Y 583.718,Z 529.66,A -85,B 0,C 180,E1 1666.369,E2 1666.369} C_VEL
LIN {X 0,Y 583.72,Z 529.66,A -85,B 0,C 180,E1 1671.653,E2 1671.653} C_VEL
LIN {X 0,Y 583.583,Z 529.66,A -85,B 0,C 180,E1 1677.112,E2 1677.112} C_VEL
LIN {X 0,Y 583.512,Z 529.66,A -85,B 0,C 180,E1 1682.259,E2 1682.259} C_VEL
LIN {X 0,Y 583.486,Z 529.66,A -85,B 0,C 180,E1 1683.395,E2 1683.395} C_VEL
LIN {X 0,Y 586.895,Z 542.193,A -85,B 0,C 180,E1 1683.745,E2 1683.745} C_VEL
LIN {X 0,Y 586.889,Z 593.278,A -85,B 0,C 180,E1 1684.581,E2 1684.581} C_VEL
LIN {X 0,Y 586.506,Z 628.915,A -85,B 0,C 180,E1 1685.741,E2 1685.741} C_VEL
LIN {X 0,Y 585.994,Z 662.234,A -85,B 0,C 180,E1 1687.395,E2 1687.395} C_VEL
LIN {X 0,Y 585.417,Z 694.604,A -85,B 0,C 180,E1 1689.637,E2 1689.637} C_VEL
LIN {X 0,Y 584.852,Z 724.023,A -85,B 0,C 180,E1 1692.405,E2 1692.405} C_VEL
LIN {X 0,Y 584.476,Z 748.039,A -85,B 0,C 180,E1 1695.427,E2 1695.427} C_VEL
LIN {X 0,Y 584.249,Z 766.703,A -85,B 0,C 180,E1 1698.594,E2 1698.594} C_VEL
LIN {X 0,Y 584.138,Z 781.541,A -85,B 0,C 180,E1 1702.206,E2 1702.206} C_VEL
LIN {X 0,Y 584.044,Z 789.994,A -85,B 0,C 180,E1 1705.555,E2 1705.555} C_VEL
LIN {X 0,Y 584.062,Z 793.512,A -85,B 0,C 180,E1 1708.52,E2 1708.52} C_VEL
LIN {X 0,Y 584.213,Z 793.511,A -85,B 0,C 180,E1 1711.481,E2 1711.481} C_VEL
LIN {X 0,Y 584.136,Z 789.992,A -85,B 0,C 180,E1 1714.445,E2 1714.445} C_VEL
LIN {X 0,Y 584.22,Z 780.272,A -85,B 0,C 180,E1 1718.168,E2 1718.168} C_VEL
LIN {X 0,Y 584.262,Z 765.275,A -85,B 0,C 180,E1 1721.682,E2 1721.682} C_VEL
LIN {X 0,Y 584.535,Z 745.324,A -85,B 0,C 180,E1 1724.961,E2 1724.961} C_VEL
LIN {X 0,Y 584.949,Z 719.939,A -85,B 0,C 180,E1 1728.034,E2 1728.034} C_VEL
LIN {X 0,Y 585.497,Z 690.847,A -85,B 0,C 180,E1 1730.657,E2 1730.657} C_VEL
LIN {X 0,Y 586.082,Z 657.723,A -85,B 0,C 180,E1 1732.868,E2 1732.868} C_VEL
LIN {X 0,Y 586.594,Z 622.68,A -85,B 0,C 180,E1 1734.508,E2 1734.508} C_VEL
LIN {X 0,Y 586.987,Z 586.864,A -85,B 0,C 180,E1 1735.564,E2 1735.564} C_VEL
LIN {X 0,Y 586.155,Z 537.627,A -85,B 0,C 180,E1 1736.351,E2 1736.351} C_VEL
LIN {X 0,Y 583.485,Z 529.66,A -85,B 0,C 180,E1 1736.637,E2 1736.637} C_VEL
LIN {X 0,Y 583.609,Z 529.66,A -85,B 0,C 180,E1 1741.438,E2 1741.438} C_VEL
LIN {X 0,Y 583.838,Z 529.66,A -85,B 0,C 180,E1 1746.757,E2 1746.757} C_VEL
LIN {X 0,Y 583.58,Z 529.66,A -85,B 0,C 180,E1 1752.245,E2 1752.245} C_VEL
LIN {X 0,Y 583.731,Z 529.66,A -85,B 0,C 180,E1 1757.772,E2 1757.772} C_VEL
LIN {X 0,Y 583.738,Z 529.66,A -85,B 0,C 180,E1 1763.522,E2 1763.522} C_VEL
LIN {X 0,Y 583.67,Z 529.66,A -85,B 0,C 180,E1 1768.867,E2 1768.867} C_VEL
LIN {X 0,Y 583.832,Z 529.66,A -85,B 0,C 180,E1 1774.774,E2 1774.774} C_VEL
LIN {X 0,Y 583.906,Z 529.66,A -85,B 0,C 180,E1 1780.371,E2 1780.371} C_VEL
LIN {X 0,Y 583.65,Z 529.66,A -85,B 0,C 180,E1 1785.019,E2 1785.019} C_VEL
LIN {X 0,Y 583.932,Z 529.66,A -85,B 0,C 180,E1 1789.58,E2 1789.58} C_VEL
LIN {X 0,Y 584.129,Z 529.66,A -85,B 0,C 180,E1 1794.071,E2 1794.071} C_VEL
LIN {X 0,Y 583.909,Z 529.66,A -85,B 0,C 180,E1 1800.002,E2 1800.002} C_VEL
LIN {X 0,Y 583.935,Z 529.66,A -85,B 0,C 180,E1 1804.448,E2 1804.448} C_VEL
LIN {X 0,Y 583.938,Z 529.66,A -85,B 0,C 180,E1 1808.922,E2 1808.922} C_VEL
LIN {X 0,Y 584.002,Z 529.66,A -85,B 0,C 180,E1 1813.449,E2 1813.449} C_VEL
LIN {X 0,Y 583.938,Z 529.66,A -85,B 0,C 180,E1 1818.067,E2 1818.067} C_VEL
LIN {X 0,Y 583.82,Z 529.66,A -85,B 0,C 180,E1 1822.813,E2 1822.813} C_VEL
LIN {X 0,Y 583.684,Z 529.66,A -85,B 0,C 180,E1 1828.477,E2 1828.477} C_VEL
LIN {X 0,Y 583.734,Z 529.66,A -85,B 0,C 180,E1 1834.663,E2 1834.663} C_VEL
LIN {X 0,Y 583.582,Z 529.66,A -85,B 0,C 180,E1 1840.275,E2 1840.275} C_VEL
LIN {X 0,Y 583.695,Z 529.66,A -85,B 0,C 180,E1 1846.377,E2 1846.377} C_VEL
LIN {X 0,Y 583.832,Z 529.943,A -85,B 0,C 180,E1 1848.655,E2 1848.655} C_VEL
LIN {X 0,Y 585.326,Z 555.193,A -85,B 0,C 180,E1 1849.014,E2 1849.014} C_VEL
LIN {X 0,Y 585.22,Z 623.775,A -85,B 0,C 180,E1 1849.959,E2 1849.959} C_VEL
LIN {X 0,Y 585.03,Z 652.966,A -85,B 0,C 180,E1 1850.959,E2 1850.959} C_VEL
LIN {X 0,Y 584.76,Z 679.161,A -85,B 0,C 180,E1 1852.479,E2 1852.479} C_VEL
LIN {X 0,Y 584.485,Z 701.745,A -85,B 0,C 180,E1 1854.453,E2 1854.453} C_VEL
LIN {X 0,Y 584.308,Z 719.694,A -85,B 0,C 180,E1 1856.746,E2 1856.746} C_VEL
LIN {X 0,Y 584.271,Z 732.75,A -85,B 0,C 180,E1 1859.259,E2 1859.259} C_VEL
LIN {X 0,Y 584.235,Z 739.761,A -85,B 0,C 180,E1 1861.425,E2 1861.425} C_VEL
LIN {X 0,Y 584.139,Z 743.629,A -85,B 0,C 180,E1 1863.949,E2 1863.949} C_VEL
LIN {X 0,Y 584.117,Z 743.864,A -85,B 0,C 180,E1 1865.585,E2 1865.585} C_VEL
LIN {X 0,Y 584.185,Z 739.919,A -85,B 0,C 180,E1 1868.424,E2 1868.424} C_VEL
LIN {X 0,Y 584.229,Z 730.565,A -85,B 0,C 180,E1 1871.163,E2 1871.163} C_VEL
LIN {X 0,Y 584.408,Z 716.15,A -85,B 0,C 180,E1 1873.691,E2 1873.691} C_VEL
LIN {X 0,Y 584.616,Z 696.464,A -85,B 0,C 180,E1 1875.99,E2 1875.99} C_VEL
LIN {X 0,Y 584.836,Z 672.258,A -85,B 0,C 180,E1 1877.898,E2 1877.898} C_VEL
LIN {X 0,Y 585.067,Z 645.131,A -85,B 0,C 180,E1 1879.284,E2 1879.284} C_VEL
LIN {X 0,Y 585.268,Z 615.779,A -85,B 0,C 180,E1 1880.117,E2 1880.117} C_VEL
LIN {X 0,Y 584.169,Z 531.635,A -85,B 0,C 180,E1 1881.224,E2 1881.224} C_VEL
LIN {X 0,Y 583.892,Z 529.66,A -85,B 0,C 180,E1 1881.266,E2 1881.266} C_VEL
LIN {X 0,Y 584.043,Z 529.66,A -85,B 0,C 180,E1 1887.037,E2 1887.037} C_VEL
LIN {X 0,Y 584.155,Z 529.66,A -85,B 0,C 180,E1 1891.48,E2 1891.48} C_VEL
LIN {X 0,Y 584.179,Z 529.66,A -85,B 0,C 180,E1 1895.93,E2 1895.93} C_VEL
LIN {X 0,Y 583.774,Z 529.66,A -85,B 0,C 180,E1 1901.934,E2 1901.934} C_VEL
LIN {X 0,Y 583.712,Z 529.66,A -85,B 0,C 180,E1 1906.955,E2 1906.955} C_VEL
LIN {X 0,Y 583.743,Z 529.66,A -85,B 0,C 180,E1 1911.466,E2 1911.466} C_VEL
LIN {X 0,Y 583.761,Z 529.66,A -85,B 0,C 180,E1 1916.067,E2 1916.067} C_VEL
LIN {X 0,Y 583.588,Z 529.66,A -85,B 0,C 180,E1 1921.427,E2 1921.427} C_VEL
LIN {X 0,Y 583.859,Z 529.66,A -85,B 0,C 180,E1 1926.753,E2 1926.753} C_VEL
LIN {X 0,Y 583.575,Z 529.66,A -85,B 0,C 180,E1 1932.244,E2 1932.244} C_VEL
LIN {X 0,Y 583.743,Z 529.66,A -85,B 0,C 180,E1 1937.768,E2 1937.768} C_VEL
LIN {X 0,Y 583.705,Z 529.66,A -85,B 0,C 180,E1 1943.514,E2 1943.514} C_VEL
LIN {X 0,Y 583.636,Z 529.66,A -85,B 0,C 180,E1 1948.86,E2 1948.86} C_VEL
LIN {X 0,Y 583.899,Z 529.66,A -85,B 0,C 180,E1 1954.757,E2 1954.757} C_VEL
LIN {X 0,Y 583.996,Z 529.66,A -85,B 0,C 180,E1 1957.644,E2 1957.644} C_VEL
LIN {X 0,Y 586.28,Z 540.374,A -85,B 0,C 180,E1 1957.907,E2 1957.907} C_VEL
LIN {X 0,Y 586.133,Z 578.744,A -85,B 0,C 180,E1 1958.598,E2 1958.598} C_VEL
LIN {X 0,Y 585.777,Z 612.962,A -85,B 0,C 180,E1 1959.836,E2 1959.836} C_VEL
LIN {X 0,Y 585.31,Z 644.333,A -85,B 0,C 180,E1 1961.588,E2 1961.588} C_VEL
LIN {X 0,Y 584.85,Z 673.268,A -85,B 0,C 180,E1 1963.895,E2 1963.895} C_VEL
LIN {X 0,Y 584.504,Z 697.497,A -85,B 0,C 180,E1 1966.563,E2 1966.563} C_VEL
LIN {X 0,Y 584.254,Z 717.269,A -85,B 0,C 180,E1 1969.582,E2 1969.582} C_VEL
LIN {X 0,Y 584.17,Z 730.939,A -85,B 0,C 180,E1 1972.616,E2 1972.616} C_VEL
LIN {X 0,Y 584.129,Z 739.353,A -85,B 0,C 180,E1 1975.553,E2 1975.553} C_VEL
LIN {X 0,Y 584.086,Z 743.468,A -85,B 0,C 180,E1 1978.518,E2 1978.518} C_VEL
LIN {X 0,Y 584.225,Z 743.409,A -85,B 0,C 180,E1 1981.478,E2 1981.478} C_VEL
LIN {X 0,Y 584.197,Z 739.174,A -85,B 0,C 180,E1 1984.442,E2 1984.442} C_VEL
LIN {X 0,Y 584.142,Z 736.694,A -85,B 0,C 180,E1 1985.472,E2 1985.472} C_VEL
LIN {X 0,Y 580.283,Z 732.015,A -85,B 0,C 180,E1 1987.092,E2 1987.092} C_VEL
LIN {X 0,Y 576.352,Z 725.896,A -85,B 0,C 180,E1 1988.684,E2 1988.684} C_VEL
LIN {X 0,Y 576.539,Z 709.001,A -85,B 0,C 180,E1 1991.881,E2 1991.881} C_VEL
LIN {X 0,Y 576.926,Z 687.18,A -85,B 0,C 180,E1 1994.788,E2 1994.788} C_VEL
LIN {X 0,Y 577.45,Z 660.251,A -85,B 0,C 180,E1 1997.385,E2 1997.385} C_VEL
LIN {X 0,Y 577.999,Z 630.426,A -85,B 0,C 180,E1 1999.44,E2 1999.44} C_VEL
LIN {X 0,Y 578.578,Z 596.941,A -85,B 0,C 180,E1 2001.012,E2 2001.012} C_VEL
LIN {X 0,Y 578.987,Z 563.793,A -85,B 0,C 180,E1 2001.941,E2 2001.941} C_VEL
LIN {X 0,Y 578.042,Z 536.06,A -85,B 0,C 180,E1 2002.391,E2 2002.391} C_VEL
LIN {X 0,Y 576.158,Z 529.66,A -85,B 0,C 180,E1 2002.606,E2 2002.606} C_VEL
LIN {X 0,Y 575.855,Z 529.66,A -85,B 0,C 180,E1 2008.141,E2 2008.141} C_VEL
LIN {X 0,Y 575.879,Z 529.66,A -85,B 0,C 180,E1 2013.383,E2 2013.383} C_VEL
LIN {X 0,Y 575.69,Z 529.66,A -85,B 0,C 180,E1 2018.979,E2 2018.979} C_VEL
LIN {X 0,Y 575.735,Z 529.66,A -85,B 0,C 180,E1 2025.042,E2 2025.042} C_VEL
LIN {X 0,Y 575.77,Z 529.66,A -85,B 0,C 180,E1 2031.025,E2 2031.025} C_VEL
LIN {X 0,Y 575.684,Z 529.66,A -85,B 0,C 180,E1 2036.603,E2 2036.603} C_VEL
LIN {X 0,Y 575.643,Z 529.66,A -85,B 0,C 180,E1 2041.846,E2 2041.846} C_VEL
LIN {X 0,Y 575.637,Z 530.379,A -85,B 0,C 180,E1 2043.029,E2 2043.029} C_VEL
LIN {X 0,Y 579.857,Z 543.555,A -85,B 0,C 180,E1 2043.42,E2 2043.42} C_VEL
LIN {X 0,Y 579.796,Z 592.139,A -85,B 0,C 180,E1 2044.217,E2 2044.217} C_VEL
LIN {X 0,Y 579.257,Z 627.739,A -85,B 0,C 180,E1 2045.368,E2 2045.368} C_VEL
LIN {X 0,Y 578.589,Z 661.83,A -85,B 0,C 180,E1 2047.065,E2 2047.065} C_VEL
LIN {X 0,Y 577.873,Z 694.617,A -85,B 0,C 180,E1 2049.36,E2 2049.36} C_VEL
LIN {X 0,Y 577.205,Z 723.356,A -85,B 0,C 180,E1 2052.089,E2 2052.089} C_VEL
LIN {X 0,Y 576.677,Z 748.139,A -85,B 0,C 180,E1 2055.24,E2 2055.24} C_VEL
LIN {X 0,Y 576.38,Z 767.43,A -85,B 0,C 180,E1 2058.579,E2 2058.579} C_VEL
LIN {X 0,Y 576.255,Z 781.541,A -85,B 0,C 180,E1 2062.099,E2 2062.099} C_VEL
LIN {X 0,Y 576.151,Z 789.993,A -85,B 0,C 180,E1 2065.494,E2 2065.494} C_VEL
LIN {X 0,Y 576.161,Z 793.512,A -85,B 0,C 180,E1 2068.5,E2 2068.5} C_VEL
LIN {X 0,Y 576.311,Z 793.511,A -85,B 0,C 180,E1 2071.501,E2 2071.501} C_VEL
LIN {X 0,Y 576.226,Z 789.992,A -85,B 0,C 180,E1 2074.507,E2 2074.507} C_VEL
LIN {X 0,Y 576.324,Z 780.271,A -85,B 0,C 180,E1 2078.28,E2 2078.28} C_VEL
LIN {X 0,Y 576.389,Z 765.07,A -85,B 0,C 180,E1 2081.884,E2 2081.884} C_VEL
LIN {X 0,Y 576.769,Z 745.326,A -85,B 0,C 180,E1 2085.167,E2 2085.167} C_VEL
LIN {X 0,Y 577.27,Z 719.939,A -85,B 0,C 180,E1 2088.282,E2 2088.282} C_VEL
LIN {X 0,Y 577.973,Z 690.102,A -85,B 0,C 180,E1 2090.999,E2 2090.999} C_VEL
LIN {X 0,Y 578.73,Z 656.492,A -85,B 0,C 180,E1 2093.248,E2 2093.248} C_VEL
LIN {X 0,Y 579.401,Z 620.606,A -85,B 0,C 180,E1 2094.91,E2 2094.91} C_VEL
LIN {X 0,Y 579.919,Z 584.764,A -85,B 0,C 180,E1 2095.943,E2 2095.943} C_VEL
LIN {X 0,Y 579.399,Z 540.634,A -85,B 0,C 180,E1 2096.642,E2 2096.642} C_VEL
LIN {X 0,Y 575.629,Z 529.66,A -85,B 0,C 180,E1 2097.058,E2 2097.058} C_VEL
LIN {X 0,Y 575.698,Z 529.66,A -85,B 0,C 180,E1 2101.617,E2 2101.617} C_VEL
LIN {X 0,Y 575.927,Z 529.66,A -85,B 0,C 180,E1 2107.059,E2 2107.059} C_VEL
LIN {X 0,Y 575.677,Z 529.66,A -85,B 0,C 180,E1 2112.964,E2 2112.964} C_VEL
LIN {X 0,Y 575.799,Z 529.66,A -85,B 0,C 180,E1 2119.071,E2 2119.071} C_VEL
LIN {X 0,Y 575.7,Z 529.66,A -85,B 0,C 180,E1 2124.788,E2 2124.788} C_VEL
LIN {X 0,Y 575.742,Z 529.66,A -85,B 0,C 180,E1 2130.136,E2 2130.136} C_VEL
LIN {X 0,Y 575.878,Z 529.66,A -85,B 0,C 180,E1 2135.215,E2 2135.215} C_VEL
LIN {X 0,Y 575.99,Z 529.66,A -85,B 0,C 180,E1 2140.587,E2 2140.587} C_VEL
LIN {X 0,Y 575.787,Z 529.66,A -85,B 0,C 180,E1 2144.809,E2 2144.809} C_VEL
LIN {X 0,Y 575.886,Z 529.66,A -85,B 0,C 180,E1 2150.957,E2 2150.957} C_VEL
LIN {X 0,Y 575.942,Z 529.66,A -85,B 0,C 180,E1 2155.494,E2 2155.494} C_VEL
LIN {X 0,Y 576.008,Z 529.66,A -85,B 0,C 180,E1 2160.002,E2 2160.002} C_VEL
LIN {X 0,Y 576.019,Z 529.66,A -85,B 0,C 180,E1 2164.51,E2 2164.51} C_VEL
LIN {X 0,Y 576.019,Z 529.66,A -85,B 0,C 180,E1 2169.045,E2 2169.045} C_VEL
LIN {X 0,Y 575.932,Z 529.66,A -85,B 0,C 180,E1 2174.201,E2 2174.201} C_VEL
LIN {X 0,Y 575.854,Z 529.66,A -85,B 0,C 180,E1 2179.919,E2 2179.919} C_VEL
LIN {X 0,Y 575.731,Z 529.66,A -85,B 0,C 180,E1 2184.796,E2 2184.796} C_VEL
LIN {X 0,Y 575.655,Z 529.66,A -85,B 0,C 180,E1 2190.111,E2 2190.111} C_VEL
LIN {X 0,Y 575.699,Z 529.66,A -85,B 0,C 180,E1 2195.217,E2 2195.217} C_VEL
LIN {X 0,Y 575.633,Z 529.66,A -85,B 0,C 180,E1 2200.949,E2 2200.949} C_VEL
LIN {X 0,Y 575.842,Z 529.66,A -85,B 0,C 180,E1 2207.203,E2 2207.203} C_VEL
LIN {X 0,Y 575.981,Z 529.66,A -85,B 0,C 180,E1 2208.416,E2 2208.416} C_VEL
LIN {X 0,Y 577.727,Z 550.883,A -85,B 0,C 180,E1 2208.744,E2 2208.744} C_VEL
LIN {X 0,Y 577.593,Z 624.369,A -85,B 0,C 180,E1 2209.77,E2 2209.77} C_VEL
LIN {X 0,Y 577.325,Z 653.15,A -85,B 0,C 180,E1 2210.777,E2 2210.777} C_VEL
LIN {X 0,Y 576.999,Z 679.572,A -85,B 0,C 180,E1 2212.338,E2 2212.338} C_VEL
LIN {X 0,Y 576.651,Z 702.276,A -85,B 0,C 180,E1 2214.366,E2 2214.366} C_VEL
LIN {X 0,Y 576.441,Z 719.807,A -85,B 0,C 180,E1 2216.651,E2 2216.651} C_VEL
LIN {X 0,Y 576.397,Z 732.579,A -85,B 0,C 180,E1 2219.138,E2 2219.138} C_VEL
LIN {X 0,Y 576.299,Z 740.861,A -85,B 0,C 180,E1 2221.88,E2 2221.88} C_VEL
LIN {X 0,Y 576.264,Z 743.367,A -85,B 0,C 180,E1 2223.566,E2 2223.566} C_VEL
LIN {X 0,Y 576.198,Z 743.267,A -85,B 0,C 180,E1 2226.438,E2 2226.438} C_VEL
LIN {X 0,Y 576.328,Z 737.716,A -85,B 0,C 180,E1 2229.3,E2 2229.3} C_VEL
LIN {X 0,Y 576.447,Z 726.199,A -85,B 0,C 180,E1 2232.15,E2 2232.15} C_VEL
LIN {X 0,Y 576.622,Z 710.069,A -85,B 0,C 180,E1 2234.634,E2 2234.634} C_VEL
LIN {X 0,Y 576.895,Z 688.499,A -85,B 0,C 180,E1 2236.865,E2 2236.865} C_VEL
LIN {X 0,Y 577.228,Z 664.474,A -85,B 0,C 180,E1 2238.547,E2 2238.547} C_VEL
LIN {X 0,Y 577.545,Z 636.467,A -85,B 0,C 180,E1 2239.794,E2 2239.794} C_VEL
LIN {X 0,Y 577.665,Z 606.729,A -85,B 0,C 180,E1 2240.461,E2 2240.461} C_VEL
LIN {X 0,Y 576.647,Z 532.891,A -85,B 0,C 180,E1 2241.426,E2 2241.426} C_VEL
LIN {X 0,Y 575.92,Z 529.66,A -85,B 0,C 180,E1 2241.496,E2 2241.496} C_VEL
LIN {X 0,Y 576.129,Z 529.66,A -85,B 0,C 180,E1 2246.997,E2 2246.997} C_VEL
LIN {X 0,Y 576.245,Z 529.66,A -85,B 0,C 180,E1 2251.5,E2 2251.5} C_VEL
LIN {X 0,Y 576.252,Z 529.66,A -85,B 0,C 180,E1 2256.012,E2 2256.012} C_VEL
LIN {X 0,Y 575.844,Z 529.66,A -85,B 0,C 180,E1 2262.101,E2 2262.101} C_VEL
LIN {X 0,Y 575.864,Z 529.66,A -85,B 0,C 180,E1 2266.752,E2 2266.752} C_VEL
LIN {X 0,Y 575.849,Z 529.66,A -85,B 0,C 180,E1 2271.522,E2 2271.522} C_VEL
LIN {X 0,Y 575.685,Z 529.66,A -85,B 0,C 180,E1 2276.971,E2 2276.971} C_VEL
LIN {X 0,Y 575.68,Z 529.66,A -85,B 0,C 180,E1 2281.617,E2 2281.617} C_VEL
LIN {X 0,Y 575.949,Z 529.66,A -85,B 0,C 180,E1 2287.056,E2 2287.056} C_VEL
LIN {X 0,Y 575.682,Z 529.66,A -85,B 0,C 180,E1 2292.961,E2 2292.961} C_VEL
LIN {X 0,Y 575.806,Z 529.66,A -85,B 0,C 180,E1 2299.066,E2 2299.066} C_VEL
LIN {X 0,Y 575.667,Z 529.66,A -85,B 0,C 180,E1 2304.78,E2 2304.78} C_VEL
LIN {X 0,Y 575.72,Z 529.66,A -85,B 0,C 180,E1 2310.13,E2 2310.13} C_VEL
LIN {X 0,Y 576.013,Z 529.66,A -85,B 0,C 180,E1 2315.217,E2 2315.217} C_VEL
LIN {X 0,Y 576.052,Z 529.66,A -85,B 0,C 180,E1 2317.321,E2 2317.321} C_VEL
LIN {X 0,Y 578.999,Z 542.098,A -85,B 0,C 180,E1 2317.637,E2 2317.637} C_VEL
LIN {X 0,Y 578.744,Z 579.804,A -85,B 0,C 180,E1 2318.342,E2 2318.342} C_VEL
LIN {X 0,Y 578.299,Z 613.654,A -85,B 0,C 180,E1 2319.597,E2 2319.597} C_VEL
LIN {X 0,Y 577.703,Z 645.749,A -85,B 0,C 180,E1 2321.435,E2 2321.435} C_VEL
LIN {X 0,Y 577.128,Z 674.305,A -85,B 0,C 180,E1 2323.771,E2 2323.771} C_VEL
LIN {X 0,Y 576.703,Z 698.957,A -85,B 0,C 180,E1 2326.57,E2 2326.57} C_VEL
LIN {X 0,Y 576.405,Z 717.263,A -85,B 0,C 180,E1 2329.439,E2 2329.439} C_VEL
LIN {X 0,Y 576.293,Z 731.301,A -85,B 0,C 180,E1 2332.617,E2 2332.617} C_VEL
LIN {X 0,Y 576.234,Z 739.355,A -85,B 0,C 180,E1 2335.492,E2 2335.492} C_VEL
LIN {X 0,Y 576.186,Z 743.469,A -85,B 0,C 180,E1 2338.497,E2 2338.497} C_VEL
LIN {X 0,Y 576.322,Z 743.411,A -85,B 0,C 180,E1 2341.498,E2 2341.498} C_VEL
LIN {X 0,Y 576.291,Z 739.178,A -85,B 0,C 180,E1 2344.503,E2 2344.503} C_VEL
LIN {X 0,Y 576.351,Z 729.084,A -85,B 0,C 180,E1 2347.898,E2 2347.898} C_VEL
LIN {X 0,Y 576.352,Z 725.896,A -85,B 0,C 180,E1 2348.684,E2 2348.684} C_VEL
LIN {X 0,Y 572.493,Z 718.86,A -85,B 0,C 180,E1 2350.242,E2 2350.242} C_VEL
LIN {X 0,Y 568.705,Z 710.763,A -85,B 0,C 180,E1 2351.763,E2 2351.763} C_VEL
LIN {X 0,Y 569.142,Z 689.031,A -85,B 0,C 180,E1 2354.784,E2 2354.784} C_VEL
LIN {X 0,Y 569.705,Z 662.975,A -85,B 0,C 180,E1 2357.394,E2 2357.394} C_VEL
LIN {X 0,Y 570.445,Z 632.319,A -85,B 0,C 180,E1 2359.596,E2 2359.596} C_VEL
LIN {X 0,Y 571.154,Z 599.629,A -85,B 0,C 180,E1 2361.198,E2 2361.198} C_VEL
LIN {X 0,Y 571.648,Z 566.854,A -85,B 0,C 180,E1 2362.174,E2 2362.174} C_VEL
LIN {X 0,Y 570.73,Z 537.851,A -85,B 0,C 180,E1 2362.671,E2 2362.671} C_VEL
LIN {X 0,Y 568.163,Z 529.66,A -85,B 0,C 180,E1 2362.938,E2 2362.938} C_VEL
LIN {X 0,Y 567.849,Z 529.66,A -85,B 0,C 180,E1 2368.727,E2 2368.727} C_VEL
LIN {X 0,Y 567.796,Z 529.66,A -85,B 0,C 180,E1 2374.528,E2 2374.528} C_VEL
LIN {X 0,Y 567.745,Z 529.66,A -85,B 0,C 180,E1 2379.631,E2 2379.631} C_VEL
LIN {X 0,Y 567.773,Z 529.66,A -85,B 0,C 180,E1 2385.852,E2 2385.852} C_VEL
LIN {X 0,Y 567.848,Z 529.66,A -85,B 0,C 180,E1 2390.407,E2 2390.407} C_VEL
LIN {X 0,Y 567.754,Z 529.66,A -85,B 0,C 180,E1 2395.475,E2 2395.475} C_VEL
LIN {X 0,Y 567.845,Z 529.66,A -85,B 0,C 180,E1 2399.676,E2 2399.676} C_VEL
LIN {X 0,Y 567.764,Z 530.379,A -85,B 0,C 180,E1 2402.624,E2 2402.624} C_VEL
LIN {X 0,Y 572.812,Z 544.294,A -85,B 0,C 180,E1 2403.077,E2 2403.077} C_VEL
LIN {X 0,Y 572.661,Z 592.589,A -85,B 0,C 180,E1 2403.884,E2 2403.884} C_VEL
LIN {X 0,Y 572.005,Z 628.987,A -85,B 0,C 180,E1 2405.088,E2 2405.088} C_VEL
LIN {X 0,Y 571.158,Z 664.089,A -85,B 0,C 180,E1 2406.888,E2 2406.888} C_VEL
LIN {X 0,Y 570.285,Z 696.983,A -85,B 0,C 180,E1 2409.274,E2 2409.274} C_VEL
LIN {X 0,Y 569.464,Z 725.679,A -85,B 0,C 180,E1 2412.103,E2 2412.103} C_VEL
LIN {X 0,Y 568.857,Z 749.909,A -85,B 0,C 180,E1 2415.296,E2 2415.296} C_VEL
LIN {X 0,Y 568.546,Z 767.911,A -85,B 0,C 180,E1 2418.519,E2 2418.519} C_VEL
LIN {X 0,Y 568.388,Z 781.541,A -85,B 0,C 180,E1 2421.989,E2 2421.989} C_VEL
LIN {X 0,Y 568.274,Z 789.993,A -85,B 0,C 180,E1 2425.432,E2 2425.432} C_VEL
LIN {X 0,Y 568.287,Z 793.512,A -85,B 0,C 180,E1 2428.479,E2 2428.479} C_VEL
LIN {X 0,Y 568.427,Z 793.511,A -85,B 0,C 180,E1 2431.522,E2 2431.522} C_VEL
LIN {X 0,Y 568.33,Z 789.991,A -85,B 0,C 180,E1 2434.569,E2 2434.569} C_VEL
LIN {X 0,Y 568.432,Z 780.271,A -85,B 0,C 180,E1 2438.396,E2 2438.396} C_VEL
LIN {X 0,Y 568.546,Z 765.908,A -85,B 0,C 180,E1 2441.885,E2 2441.885} C_VEL
LIN {X 0,Y 568.965,Z 746.659,A -85,B 0,C 180,E1 2445.184,E2 2445.184} C_VEL
LIN {X 0,Y 569.578,Z 721.559,A -85,B 0,C 180,E1 2448.364,E2 2448.364} C_VEL
LIN {X 0,Y 570.396,Z 692.099,A -85,B 0,C 180,E1 2451.129,E2 2451.129} C_VEL
LIN {X 0,Y 571.258,Z 660.241,A -85,B 0,C 180,E1 2453.343,E2 2453.343} C_VEL
LIN {X 0,Y 572.113,Z 624.411,A -85,B 0,C 180,E1 2455.104,E2 2455.104} C_VEL
LIN {X 0,Y 572.765,Z 587.659,A -85,B 0,C 180,E1 2456.23,E2 2456.23} C_VEL
LIN {X 0,Y 572.198,Z 542.401,A -85,B 0,C 180,E1 2456.98,E2 2456.98} C_VEL
LIN {X 0,Y 567.715,Z 529.66,A -85,B 0,C 180,E1 2457.455,E2 2457.455} C_VEL
LIN {X 0,Y 567.744,Z 529.66,A -85,B 0,C 180,E1 2462.113,E2 2462.113} C_VEL
LIN {X 0,Y 568.002,Z 529.66,A -85,B 0,C 180,E1 2467.665,E2 2467.665} C_VEL
LIN {X 0,Y 567.736,Z 529.66,A -85,B 0,C 180,E1 2474.144,E2 2474.144} C_VEL
LIN {X 0,Y 567.828,Z 529.66,A -85,B 0,C 180,E1 2478.369,E2 2478.369} C_VEL
LIN {X 0,Y 567.84,Z 529.66,A -85,B 0,C 180,E1 2484.226,E2 2484.226} C_VEL
LIN {X 0,Y 567.835,Z 529.66,A -85,B 0,C 180,E1 2489.677,E2 2489.677} C_VEL
LIN {X 0,Y 567.927,Z 529.66,A -85,B 0,C 180,E1 2494.844,E2 2494.844} C_VEL
LIN {X 0,Y 568.004,Z 529.66,A -85,B 0,C 180,E1 2499.798,E2 2499.798} C_VEL
LIN {X 0,Y 567.894,Z 529.66,A -85,B 0,C 180,E1 2504.593,E2 2504.593} C_VEL
LIN {X 0,Y 567.98,Z 529.66,A -85,B 0,C 180,E1 2510.83,E2 2510.83} C_VEL
LIN {X 0,Y 568.052,Z 529.66,A -85,B 0,C 180,E1 2515.431,E2 2515.431} C_VEL
LIN {X 0,Y 568.134,Z 529.66,A -85,B 0,C 180,E1 2520.002,E2 2520.002} C_VEL
LIN {X 0,Y 568.106,Z 529.66,A -85,B 0,C 180,E1 2524.572,E2 2524.572} C_VEL
LIN {X 0,Y 568.087,Z 529.66,A -85,B 0,C 180,E1 2529.173,E2 2529.173} C_VEL
LIN {X 0,Y 568.119,Z 529.66,A -85,B 0,C 180,E1 2533.832,E2 2533.832} C_VEL
LIN {X 0,Y 568.057,Z 529.66,A -85,B 0,C 180,E1 2538.59,E2 2538.59} C_VEL
LIN {X 0,Y 567.935,Z 529.66,A -85,B 0,C 180,E1 2543.489,E2 2543.489} C_VEL
LIN {X 0,Y 567.822,Z 529.66,A -85,B 0,C 180,E1 2548.719,E2 2548.719} C_VEL
LIN {X 0,Y 567.802,Z 529.66,A -85,B 0,C 180,E1 2554.526,E2 2554.526} C_VEL
LIN {X 0,Y 567.72,Z 529.66,A -85,B 0,C 180,E1 2559.639,E2 2559.639} C_VEL
LIN {X 0,Y 567.784,Z 529.66,A -85,B 0,C 180,E1 2565.857,E2 2565.857} C_VEL
LIN {X 0,Y 568.102,Z 530.24,A -85,B 0,C 180,E1 2568.195,E2 2568.195} C_VEL
LIN {X 0,Y 570.166,Z 552.37,A -85,B 0,C 180,E1 2568.542,E2 2568.542} C_VEL
LIN {X 0,Y 569.97,Z 624.254,A -85,B 0,C 180,E1 2569.559,E2 2569.559} C_VEL
LIN {X 0,Y 569.64,Z 653.323,A -85,B 0,C 180,E1 2570.59,E2 2570.59} C_VEL
LIN {X 0,Y 569.243,Z 679.869,A -85,B 0,C 180,E1 2572.185,E2 2572.185} C_VEL
LIN {X 0,Y 568.817,Z 702.952,A -85,B 0,C 180,E1 2574.293,E2 2574.293} C_VEL
LIN {X 0,Y 568.589,Z 721.561,A -85,B 0,C 180,E1 2576.821,E2 2576.821} C_VEL
LIN {X 0,Y 568.466,Z 733.615,A -85,B 0,C 180,E1 2579.318,E2 2579.318} C_VEL
LIN {X 0,Y 568.438,Z 740.076,A -85,B 0,C 180,E1 2581.455,E2 2581.455} C_VEL
LIN {X 0,Y 568.304,Z 743.914,A -85,B 0,C 180,E1 2584.53,E2 2584.53} C_VEL
LIN {X 0,Y 568.358,Z 742.132,A -85,B 0,C 180,E1 2587.357,E2 2587.357} C_VEL
LIN {X 0,Y 568.459,Z 734.712,A -85,B 0,C 180,E1 2590.292,E2 2590.292} C_VEL
LIN {X 0,Y 568.59,Z 721.943,A -85,B 0,C 180,E1 2593.026,E2 2593.026} C_VEL
LIN {X 0,Y 568.848,Z 704.486,A -85,B 0,C 180,E1 2595.443,E2 2595.443} C_VEL
LIN {X 0,Y 569.204,Z 682.004,A -85,B 0,C 180,E1 2597.56,E2 2597.56} C_VEL
LIN {X 0,Y 569.655,Z 655.989,A -85,B 0,C 180,E1 2599.191,E2 2599.191} C_VEL
LIN {X 0,Y 569.97,Z 626.908,A -85,B 0,C 180,E1 2600.283,E2 2600.283} C_VEL
LIN {X 0,Y 570.062,Z 580.863,A -85,B 0,C 180,E1 2601.005,E2 2601.005} C_VEL
LIN {X 0,Y 568.963,Z 534.14,A -85,B 0,C 180,E1 2601.639,E2 2601.639} C_VEL
LIN {X 0,Y 567.975,Z 529.66,A -85,B 0,C 180,E1 2601.789,E2 2601.789} C_VEL
LIN {X 0,Y 568.218,Z 529.66,A -85,B 0,C 180,E1 2606.955,E2 2606.955} C_VEL
LIN {X 0,Y 568.36,Z 529.66,A -85,B 0,C 180,E1 2611.521,E2 2611.521} C_VEL
LIN {X 0,Y 568.317,Z 529.66,A -85,B 0,C 180,E1 2616.096,E2 2616.096} C_VEL
LIN {X 0,Y 567.932,Z 529.66,A -85,B 0,C 180,E1 2622.272,E2 2622.272} C_VEL
LIN {X 0,Y 567.948,Z 529.66,A -85,B 0,C 180,E1 2626.993,E2 2626.993} C_VEL
LIN {X 0,Y 567.899,Z 529.66,A -85,B 0,C 180,E1 2631.838,E2 2631.838} C_VEL
LIN {X 0,Y 567.799,Z 529.66,A -85,B 0,C 180,E1 2636.858,E2 2636.858} C_VEL
LIN {X 0,Y 567.739,Z 529.66,A -85,B 0,C 180,E1 2642.111,E2 2642.111} C_VEL
LIN {X 0,Y 568.023,Z 529.66,A -85,B 0,C 180,E1 2647.662,E2 2647.662} C_VEL
LIN {X 0,Y 567.742,Z 529.66,A -85,B 0,C 180,E1 2654.139,E2 2654.139} C_VEL
LIN {X 0,Y 567.837,Z 529.66,A -85,B 0,C 180,E1 2658.365,E2 2658.365} C_VEL
LIN {X 0,Y 567.808,Z 529.66,A -85,B 0,C 180,E1 2664.219,E2 2664.219} C_VEL
LIN {X 0,Y 567.808,Z 529.66,A -85,B 0,C 180,E1 2669.671,E2 2669.671} C_VEL
LIN {X 0,Y 568.029,Z 529.66,A -85,B 0,C 180,E1 2674.845,E2 2674.845} C_VEL
LIN {X 0,Y 568.148,Z 530.362,A -85,B 0,C 180,E1 2677.029,E2 2677.029} C_VEL
LIN {X 0,Y 571.712,Z 543.044,A -85,B 0,C 180,E1 2677.35,E2 2677.35} C_VEL
LIN {X 0,Y 571.366,Z 581.234,A -85,B 0,C 180,E1 2678.09,E2 2678.09} C_VEL
LIN {X 0,Y 570.813,Z 615.221,A -85,B 0,C 180,E1 2679.393,E2 2679.393} C_VEL
LIN {X 0,Y 570.107,Z 647.116,A -85,B 0,C 180,E1 2681.279,E2 2681.279} C_VEL
LIN {X 0,Y 569.396,Z 675.295,A -85,B 0,C 180,E1 2683.644,E2 2683.644} C_VEL
LIN {X 0,Y 568.931,Z 698.956,A -85,B 0,C 180,E1 2686.383,E2 2686.383} C_VEL
LIN {X 0,Y 568.564,Z 717.257,A -85,B 0,C 180,E1 2689.291,E2 2689.291} C_VEL
LIN {X 0,Y 568.414,Z 731.663,A -85,B 0,C 180,E1 2692.619,E2 2692.619} C_VEL
LIN {X 0,Y 568.389,Z 740.808,A -85,B 0,C 180,E1 2696.192,E2 2696.192} C_VEL
LIN {X 0,Y 568.278,Z 743.997,A -85,B 0,C 180,E1 2699.998,E2 2699.998} C_VEL
LIN {X 0,Y 568.372,Z 741.855,A -85,B 0,C 180,E1 2703.042,E2 2703.042} C_VEL
LIN {X 0,Y 568.383,Z 734.293,A -85,B 0,C 180,E1 2706.476,E2 2706.476} C_VEL
LIN {X 0,Y 568.577,Z 720.753,A -85,B 0,C 180,E1 2709.932,E2 2709.932} C_VEL
LIN {X 0,Y 568.705,Z 710.763,A -85,B 0,C 180,E1 2711.763,E2 2711.763} C_VEL
LIN {X 0,Y 564.927,Z 701.747,A -85,B 0,C 180,E1 2713.237,E2 2713.237} C_VEL
LIN {X 0,Y 561.322,Z 691.728,A -85,B 0,C 180,E1 2714.66,E2 2714.66} C_VEL
LIN {X 0,Y 562.002,Z 665.605,A -85,B 0,C 180,E1 2717.408,E2 2717.408} C_VEL
LIN {X 0,Y 562.848,Z 635.509,A -85,B 0,C 180,E1 2719.674,E2 2719.674} C_VEL
LIN {X 0,Y 563.667,Z 603.284,A -85,B 0,C 180,E1 2721.339,E2 2721.339} C_VEL
LIN {X 0,Y 564.253,Z 570.655,A -85,B 0,C 180,E1 2722.394,E2 2722.394} C_VEL
LIN {X 0,Y 563.477,Z 539.849,A -85,B 0,C 180,E1 2722.953,E2 2722.953} C_VEL
LIN {X 0,Y 560.188,Z 529.66,A -85,B 0,C 180,E1 2723.26,E2 2723.26} C_VEL
LIN {X 0,Y 559.91,Z 529.66,A -85,B 0,C 180,E1 2729.017,E2 2729.017} C_VEL
LIN {X 0,Y 559.914,Z 529.66,A -85,B 0,C 180,E1 2734.466,E2 2734.466} C_VEL
LIN {X 0,Y 559.744,Z 529.66,A -85,B 0,C 180,E1 2740.313,E2 2740.313} C_VEL
LIN {X 0,Y 559.822,Z 529.66,A -85,B 0,C 180,E1 2745.508,E2 2745.508} C_VEL
LIN {X 0,Y 559.903,Z 529.66,A -85,B 0,C 180,E1 2751.401,E2 2751.401} C_VEL
LIN {X 0,Y 559.815,Z 529.66,A -85,B 0,C 180,E1 2756.675,E2 2756.675} C_VEL
LIN {X 0,Y 559.861,Z 529.66,A -85,B 0,C 180,E1 2762.171,E2 2762.171} C_VEL
LIN {X 0,Y 565.784,Z 546.128,A -85,B 0,C 180,E1 2762.741,E2 2762.741} C_VEL
LIN {X 0,Y 565.558,Z 592.873,A -85,B 0,C 180,E1 2763.538,E2 2763.538} C_VEL
LIN {X 0,Y 564.755,Z 629.008,A -85,B 0,C 180,E1 2764.747,E2 2764.747} C_VEL
LIN {X 0,Y 563.789,Z 663.505,A -85,B 0,C 180,E1 2766.531,E2 2766.531} C_VEL
LIN {X 0,Y 562.721,Z 696.982,A -85,B 0,C 180,E1 2768.983,E2 2768.983} C_VEL
LIN {X 0,Y 561.808,Z 724.998,A -85,B 0,C 180,E1 2771.772,E2 2771.772} C_VEL
LIN {X 0,Y 561.089,Z 749.569,A -85,B 0,C 180,E1 2775.036,E2 2775.036} C_VEL
LIN {X 0,Y 560.695,Z 767.908,A -85,B 0,C 180,E1 2778.356,E2 2778.356} C_VEL
LIN {X 0,Y 560.532,Z 781.541,A -85,B 0,C 180,E1 2781.876,E2 2781.876} C_VEL
LIN {X 0,Y 560.383,Z 789.992,A -85,B 0,C 180,E1 2785.367,E2 2785.367} C_VEL
LIN {X 0,Y 560.386,Z 793.512,A -85,B 0,C 180,E1 2788.458,E2 2788.458} C_VEL
LIN {X 0,Y 560.524,Z 793.512,A -85,B 0,C 180,E1 2791.543,E2 2791.543} C_VEL
LIN {X 0,Y 560.41,Z 789.357,A -85,B 0,C 180,E1 2794.974,E2 2794.974} C_VEL
LIN {X 0,Y 560.557,Z 780.27,A -85,B 0,C 180,E1 2798.515,E2 2798.515} C_VEL
LIN {X 0,Y 560.679,Z 765.976,A -85,B 0,C 180,E1 2802.04,E2 2802.04} C_VEL
LIN {X 0,Y 561.188,Z 746.348,A -85,B 0,C 180,E1 2805.446,E2 2805.446} C_VEL
LIN {X 0,Y 561.906,Z 721.244,A -85,B 0,C 180,E1 2808.66,E2 2808.66} C_VEL
LIN {X 0,Y 562.901,Z 690.855,A -85,B 0,C 180,E1 2811.527,E2 2811.527} C_VEL
LIN {X 0,Y 563.949,Z 658.21,A -85,B 0,C 180,E1 2813.789,E2 2813.789} C_VEL
LIN {X 0,Y 564.987,Z 622.082,A -85,B 0,C 180,E1 2815.534,E2 2815.534} C_VEL
LIN {X 0,Y 565.684,Z 586.958,A -85,B 0,C 180,E1 2816.599,E2 2816.599} C_VEL
LIN {X 0,Y 565.252,Z 544.611,A -85,B 0,C 180,E1 2817.308,E2 2817.308} C_VEL
LIN {X 0,Y 559.837,Z 529.66,A -85,B 0,C 180,E1 2817.895,E2 2817.895} C_VEL
LIN {X 0,Y 559.761,Z 529.66,A -85,B 0,C 180,E1 2823.317,E2 2823.317} C_VEL
LIN {X 0,Y 559.964,Z 529.66,A -85,B 0,C 180,E1 2828.607,E2 2828.607} C_VEL
LIN {X 0,Y 559.805,Z 529.66,A -85,B 0,C 180,E1 2834.496,E2 2834.496} C_VEL
LIN {X 0,Y 559.844,Z 529.66,A -85,B 0,C 180,E1 2839.696,E2 2839.696} C_VEL
LIN {X 0,Y 559.834,Z 529.66,A -85,B 0,C 180,E1 2845.529,E2 2845.529} C_VEL
LIN {X 0,Y 559.869,Z 529.66,A -85,B 0,C 180,E1 2850.981,E2 2850.981} C_VEL
LIN {X 0,Y 559.945,Z 529.66,A -85,B 0,C 180,E1 2856.387,E2 2856.387} C_VEL
LIN {X 0,Y 560.118,Z 529.66,A -85,B 0,C 180,E1 2861.141,E2 2861.141} C_VEL
LIN {X 0,Y 559.824,Z 529.66,A -85,B 0,C 180,E1 2866.02,E2 2866.02} C_VEL
LIN {X 0,Y 560.074,Z 529.66,A -85,B 0,C 180,E1 2870.699,E2 2870.699} C_VEL
LIN {X 0,Y 560.163,Z 529.66,A -85,B 0,C 180,E1 2875.367,E2 2875.367} C_VEL
LIN {X 0,Y 560.233,Z 529.66,A -85,B 0,C 180,E1 2880.002,E2 2880.002} C_VEL
LIN {X 0,Y 560.195,Z 529.66,A -85,B 0,C 180,E1 2884.672,E2 2884.672} C_VEL
LIN {X 0,Y 560.173,Z 529.66,A -85,B 0,C 180,E1 2889.303,E2 2889.303} C_VEL
LIN {X 0,Y 560.152,Z 529.66,A -85,B 0,C 180,E1 2894.114,E2 2894.114} C_VEL
LIN {X 0,Y 560.047,Z 529.66,A -85,B 0,C 180,E1 2899.429,E2 2899.429} C_VEL
LIN {X 0,Y 559.977,Z 529.66,A -85,B 0,C 180,E1 2903.844,E2 2903.844} C_VEL
LIN {X 0,Y 559.883,Z 529.66,A -85,B 0,C 180,E1 2909.023,E2 2909.023} C_VEL
LIN {X 0,Y 559.921,Z 529.66,A -85,B 0,C 180,E1 2914.47,E2 2914.47} C_VEL
LIN {X 0,Y 559.74,Z 529.66,A -85,B 0,C 180,E1 2920.987,E2 2920.987} C_VEL
LIN {X 0,Y 559.92,Z 529.66,A -85,B 0,C 180,E1 2926.692,E2 2926.692} C_VEL
LIN {X 0,Y 560.146,Z 529.909,A -85,B 0,C 180,E1 2927.945,E2 2927.945} C_VEL
LIN {X 0,Y 562.595,Z 551.599,A -85,B 0,C 180,E1 2928.305,E2 2928.305} C_VEL
LIN {X 0,Y 562.385,Z 623.787,A -85,B 0,C 180,E1 2929.334,E2 2929.334} C_VEL
LIN {X 0,Y 562.013,Z 651.784,A -85,B 0,C 180,E1 2930.317,E2 2930.317} C_VEL
LIN {X 0,Y 561.553,Z 678.609,A -85,B 0,C 180,E1 2931.915,E2 2931.915} C_VEL
LIN {X 0,Y 561.077,Z 701.993,A -85,B 0,C 180,E1 2934.036,E2 2934.036} C_VEL
LIN {X 0,Y 560.716,Z 720.574,A -85,B 0,C 180,E1 2936.542,E2 2936.542} C_VEL
LIN {X 0,Y 560.61,Z 733.62,A -85,B 0,C 180,E1 2939.241,E2 2939.241} C_VEL
LIN {X 0,Y 560.496,Z 741.048,A -85,B 0,C 180,E1 2941.887,E2 2941.887} C_VEL
LIN {X 0,Y 560.43,Z 743.904,A -85,B 0,C 180,E1 2944.48,E2 2944.48} C_VEL
LIN {X 0,Y 560.46,Z 742.611,A -85,B 0,C 180,E1 2947.074,E2 2947.074} C_VEL
LIN {X 0,Y 560.574,Z 735.926,A -85,B 0,C 180,E1 2950.01,E2 2950.01} C_VEL
LIN {X 0,Y 560.707,Z 723.945,A -85,B 0,C 180,E1 2952.78,E2 2952.78} C_VEL
LIN {X 0,Y 561.007,Z 705.981,A -85,B 0,C 180,E1 2955.416,E2 2955.416} C_VEL
LIN {X 0,Y 561.426,Z 683.941,A -85,B 0,C 180,E1 2957.582,E2 2957.582} C_VEL
LIN {X 0,Y 561.944,Z 658.424,A -85,B 0,C 180,E1 2959.263,E2 2959.263} C_VEL
LIN {X 0,Y 562.315,Z 630.609,A -85,B 0,C 180,E1 2960.393,E2 2960.393} C_VEL
LIN {X 0,Y 562.443,Z 596.633,A -85,B 0,C 180,E1 2961.023,E2 2961.023} C_VEL
LIN {X 0,Y 561.68,Z 536.549,A -85,B 0,C 180,E1 2961.83,E2 2961.83} C_VEL
LIN {X 0,Y 560.038,Z 529.66,A -85,B 0,C 180,E1 2962.011,E2 2962.011} C_VEL
LIN {X 0,Y 560.303,Z 529.66,A -85,B 0,C 180,E1 2966.912,E2 2966.912} C_VEL
LIN {X 0,Y 560.449,Z 529.66,A -85,B 0,C 180,E1 2971.542,E2 2971.542} C_VEL
LIN {X 0,Y 560.395,Z 529.66,A -85,B 0,C 180,E1 2976.183,E2 2976.183} C_VEL
LIN {X 0,Y 560.007,Z 529.66,A -85,B 0,C 180,E1 2982.448,E2 2982.448} C_VEL
LIN {X 0,Y 560.014,Z 529.66,A -85,B 0,C 180,E1 2987.241,E2 2987.241} C_VEL
LIN {X 0,Y 559.947,Z 529.66,A -85,B 0,C 180,E1 2992.165,E2 2992.165} C_VEL
LIN {X 0,Y 559.832,Z 529.66,A -85,B 0,C 180,E1 2997.272,E2 2997.272} C_VEL
LIN {X 0,Y 559.768,Z 529.66,A -85,B 0,C 180,E1 3002.625,E2 3002.625} C_VEL
LIN {X 0,Y 560.006,Z 529.66,A -85,B 0,C 180,E1 3008.298,E2 3008.298} C_VEL
LIN {X 0,Y 559.811,Z 529.66,A -85,B 0,C 180,E1 3014.493,E2 3014.493} C_VEL
LIN {X 0,Y 559.851,Z 529.66,A -85,B 0,C 180,E1 3019.691,E2 3019.691} C_VEL
LIN {X 0,Y 559.799,Z 529.66,A -85,B 0,C 180,E1 3025.521,E2 3025.521} C_VEL
LIN {X 0,Y 559.845,Z 529.66,A -85,B 0,C 180,E1 3030.975,E2 3030.975} C_VEL
LIN {X 0,Y 560.213,Z 529.66,A -85,B 0,C 180,E1 3036.672,E2 3036.672} C_VEL
LIN {X 0,Y 564.418,Z 544.064,A -85,B 0,C 180,E1 3037.055,E2 3037.055} C_VEL
LIN {X 0,Y 564.026,Z 581.148,A -85,B 0,C 180,E1 3037.788,E2 3037.788} C_VEL
LIN {X 0,Y 563.389,Z 615.21,A -85,B 0,C 180,E1 3039.109,E2 3039.109} C_VEL
LIN {X 0,Y 562.524,Z 647.24,A -85,B 0,C 180,E1 3041.026,E2 3041.026} C_VEL
LIN {X 0,Y 561.718,Z 675.287,A -85,B 0,C 180,E1 3043.414,E2 3043.414} C_VEL
LIN {X 0,Y 561.137,Z 698.955,A -85,B 0,C 180,E1 3046.19,E2 3046.19} C_VEL
LIN {X 0,Y 560.752,Z 717.251,A -85,B 0,C 180,E1 3049.14,E2 3049.14} C_VEL
LIN {X 0,Y 560.535,Z 730.799,A -85,B 0,C 180,E1 3052.262,E2 3052.262} C_VEL
LIN {X 0,Y 560.458,Z 739.358,A -85,B 0,C 180,E1 3055.365,E2 3055.365} C_VEL
LIN {X 0,Y 560.411,Z 743.471,A -85,B 0,C 180,E1 3058.455,E2 3058.455} C_VEL
LIN {X 0,Y 560.534,Z 743.415,A -85,B 0,C 180,E1 3061.541,E2 3061.541} C_VEL
LIN {X 0,Y 560.464,Z 738.367,A -85,B 0,C 180,E1 3065.014,E2 3065.014} C_VEL
LIN {X 0,Y 560.613,Z 727.559,A -85,B 0,C 180,E1 3068.511,E2 3068.511} C_VEL
LIN {X 0,Y 560.853,Z 711.331,A -85,B 0,C 180,E1 3071.836,E2 3071.836} C_VEL
LIN {X 0,Y 561.322,Z 691.728,A -85,B 0,C 180,E1 3074.66,E2 3074.66} C_VEL
LIN {X 0,Y 557.699,Z 680.907,A -85,B 0,C 180,E1 3076.026,E2 3076.026} C_VEL
LIN {X 0,Y 554.25,Z 670.815,A -85,B 0,C 180,E1 3077.17,E2 3077.17} C_VEL
LIN {X 0,Y 554.24,Z 669.209,A -85,B 0,C 180,E1 3077.325,E2 3077.325} C_VEL
LIN {X 0,Y 555.196,Z 640.489,A -85,B 0,C 180,E1 3079.624,E2 3079.624} C_VEL
LIN {X 0,Y 556.189,Z 608.082,A -85,B 0,C 180,E1 3081.431,E2 3081.431} C_VEL
LIN {X 0,Y 556.892,Z 575.005,A -85,B 0,C 180,E1 3082.596,E2 3082.596} C_VEL
LIN {X 0,Y 556.442,Z 542.328,A -85,B 0,C 180,E1 3083.227,E2 3083.227} C_VEL
LIN {X 0,Y 552.191,Z 529.66,A -85,B 0,C 180,E1 3083.656,E2 3083.656} C_VEL
LIN {X 0,Y 551.968,Z 529.66,A -85,B 0,C 180,E1 3089.475,E2 3089.475} C_VEL
LIN {X 0,Y 551.954,Z 529.66,A -85,B 0,C 180,E1 3095.035,E2 3095.035} C_VEL
LIN {X 0,Y 551.868,Z 529.66,A -85,B 0,C 180,E1 3101.01,E2 3101.01} C_VEL
LIN {X 0,Y 551.959,Z 529.66,A -85,B 0,C 180,E1 3106.886,E2 3106.886} C_VEL
LIN {X 0,Y 551.984,Z 529.66,A -85,B 0,C 180,E1 3113.029,E2 3113.029} C_VEL
LIN {X 0,Y 551.934,Z 529.66,A -85,B 0,C 180,E1 3118.705,E2 3118.705} C_VEL
LIN {X 0,Y 551.957,Z 530.085,A -85,B 0,C 180,E1 3121.767,E2 3121.767} C_VEL
LIN {X 0,Y 558.81,Z 550.575,A -85,B 0,C 180,E1 3122.435,E2 3122.435} C_VEL
LIN {X 0,Y 558.445,Z 593.738,A -85,B 0,C 180,E1 3123.199,E2 3123.199} C_VEL
LIN {X 0,Y 557.561,Z 629.004,A -85,B 0,C 180,E1 3124.398,E2 3124.398} C_VEL
LIN {X 0,Y 556.43,Z 663.44,A -85,B 0,C 180,E1 3126.198,E2 3126.198} C_VEL
LIN {X 0,Y 555.233,Z 696.98,A -85,B 0,C 180,E1 3128.685,E2 3128.685} C_VEL
LIN {X 0,Y 554.149,Z 725.303,A -85,B 0,C 180,E1 3131.546,E2 3131.546} C_VEL
LIN {X 0,Y 553.364,Z 749.091,A -85,B 0,C 180,E1 3134.75,E2 3134.75} C_VEL
LIN {X 0,Y 552.856,Z 767.908,A -85,B 0,C 180,E1 3138.188,E2 3138.188} C_VEL
LIN {X 0,Y 552.685,Z 781.541,A -85,B 0,C 180,E1 3141.759,E2 3141.759} C_VEL
LIN {X 0,Y 552.509,Z 789.992,A -85,B 0,C 180,E1 3145.301,E2 3145.301} C_VEL
LIN {X 0,Y 552.488,Z 793.513,A -85,B 0,C 180,E1 3148.436,E2 3148.436} C_VEL
LIN {X 0,Y 552.621,Z 793.512,A -85,B 0,C 180,E1 3151.565,E2 3151.565} C_VEL
LIN {X 0,Y 552.538,Z 789.99,A -85,B 0,C 180,E1 3154.7,E2 3154.7} C_VEL
LIN {X 0,Y 552.665,Z 780.27,A -85,B 0,C 180,E1 3158.638,E2 3158.638} C_VEL
LIN {X 0,Y 552.822,Z 765.975,A -85,B 0,C 180,E1 3162.214,E2 3162.214} C_VEL
LIN {X 0,Y 553.388,Z 747.137,A -85,B 0,C 180,E1 3165.549,E2 3165.549} C_VEL
LIN {X 0,Y 554.23,Z 721.965,A -85,B 0,C 180,E1 3168.844,E2 3168.844} C_VEL
LIN {X 0,Y 555.356,Z 692.105,A -85,B 0,C 180,E1 3171.729,E2 3171.729} C_VEL
LIN {X 0,Y 556.559,Z 660.235,A -85,B 0,C 180,E1 3173.998,E2 3173.998} C_VEL
LIN {X 0,Y 557.699,Z 625.82,A -85,B 0,C 180,E1 3175.737,E2 3175.737} C_VEL
LIN {X 0,Y 558.57,Z 588.985,A -85,B 0,C 180,E1 3176.92,E2 3176.92} C_VEL
LIN {X 0,Y 558.189,Z 546.625,A -85,B 0,C 180,E1 3177.654,E2 3177.654} C_VEL
LIN {X 0,Y 551.953,Z 529.66,A -85,B 0,C 180,E1 3178.305,E2 3178.305} C_VEL
LIN {X 0,Y 551.858,Z 529.66,A -85,B 0,C 180,E1 3183.154,E2 3183.154} C_VEL
LIN {X 0,Y 552.02,Z 529.66,A -85,B 0,C 180,E1 3188.957,E2 3188.957} C_VEL
LIN {X 0,Y 551.924,Z 529.66,A -85,B 0,C 180,E1 3195.305,E2 3195.305} C_VEL
LIN {X 0,Y 551.957,Z 529.66,A -85,B 0,C 180,E1 3201.042,E2 3201.042} C_VEL
LIN {X 0,Y 551.889,Z 529.66,A -85,B 0,C 180,E1 3206.852,E2 3206.852} C_VEL
LIN {X 0,Y 551.974,Z 529.66,A -85,B 0,C 180,E1 3212.309,E2 3212.309} C_VEL
LIN {X 0,Y 552.014,Z 529.66,A -85,B 0,C 180,E1 3217.501,E2 3217.501} C_VEL
LIN {X 0,Y 552.223,Z 529.66,A -85,B 0,C 180,E1 3223.021,E2 3223.021} C_VEL
LIN {X 0,Y 552.182,Z 529.66,A -85,B 0,C 180,E1 3229.676,E2 3229.676} C_VEL
LIN {X 0,Y 552.265,Z 529.66,A -85,B 0,C 180,E1 3235.3,E2 3235.3} C_VEL
LIN {X 0,Y 552.335,Z 529.66,A -85,B 0,C 180,E1 3240.002,E2 3240.002} C_VEL
LIN {X 0,Y 552.316,Z 529.66,A -85,B 0,C 180,E1 3244.703,E2 3244.703} C_VEL
LIN {X 0,Y 552.146,Z 529.66,A -85,B 0,C 180,E1 3250.303,E2 3250.303} C_VEL
LIN {X 0,Y 552.097,Z 529.66,A -85,B 0,C 180,E1 3255.864,E2 3255.864} C_VEL
LIN {X 0,Y 552.062,Z 529.66,A -85,B 0,C 180,E1 3261.665,E2 3261.665} C_VEL
LIN {X 0,Y 551.955,Z 529.66,A -85,B 0,C 180,E1 3267.697,E2 3267.697} C_VEL
LIN {X 0,Y 552.029,Z 529.66,A -85,B 0,C 180,E1 3273.143,E2 3273.143} C_VEL
LIN {X 0,Y 551.789,Z 529.66,A -85,B 0,C 180,E1 3278.978,E2 3278.978} C_VEL
LIN {X 0,Y 551.894,Z 529.66,A -85,B 0,C 180,E1 3284.691,E2 3284.691} C_VEL
LIN {X 0,Y 552.169,Z 529.66,A -85,B 0,C 180,E1 3287.677,E2 3287.677} C_VEL
LIN {X 0,Y 555.034,Z 550.031,A -85,B 0,C 180,E1 3288.051,E2 3288.051} C_VEL
LIN {X 0,Y 554.773,Z 624.79,A -85,B 0,C 180,E1 3289.139,E2 3289.139} C_VEL
LIN {X 0,Y 554.309,Z 653.551,A -85,B 0,C 180,E1 3290.196,E2 3290.196} C_VEL
LIN {X 0,Y 553.793,Z 679.022,A -85,B 0,C 180,E1 3291.76,E2 3291.76} C_VEL
LIN {X 0,Y 553.283,Z 702.175,A -85,B 0,C 180,E1 3293.901,E2 3293.901} C_VEL
LIN {X 0,Y 552.876,Z 720.801,A -85,B 0,C 180,E1 3296.461,E2 3296.461} C_VEL
LIN {X 0,Y 552.725,Z 733.254,A -85,B 0,C 180,E1 3299.063,E2 3299.063} C_VEL
LIN {X 0,Y 552.619,Z 740.608,A -85,B 0,C 180,E1 3301.619,E2 3301.619} C_VEL
LIN {X 0,Y 552.527,Z 743.872,A -85,B 0,C 180,E1 3304.327,E2 3304.327} C_VEL
LIN {X 0,Y 552.583,Z 741.986,A -85,B 0,C 180,E1 3307.522,E2 3307.522} C_VEL
LIN {X 0,Y 552.717,Z 734.52,A -85,B 0,C 180,E1 3310.502,E2 3310.502} C_VEL
LIN {X 0,Y 552.84,Z 722.507,A -85,B 0,C 180,E1 3313.156,E2 3313.156} C_VEL
LIN {X 0,Y 553.167,Z 706.02,A -85,B 0,C 180,E1 3315.562,E2 3315.562} C_VEL
LIN {X 0,Y 553.655,Z 683.772,A -85,B 0,C 180,E1 3317.776,E2 3317.776} C_VEL
LIN {X 0,Y 554.262,Z 657.618,A -85,B 0,C 180,E1 3319.509,E2 3319.509} C_VEL
LIN {X 0,Y 554.727,Z 629.002,A -85,B 0,C 180,E1 3320.655,E2 3320.655} C_VEL
LIN {X 0,Y 554.896,Z 592.723,A -85,B 0,C 180,E1 3321.299,E2 3321.299} C_VEL
LIN {X 0,Y 554.115,Z 537.826,A -85,B 0,C 180,E1 3322.05,E2 3322.05} C_VEL
LIN {X 0,Y 552.032,Z 529.66,A -85,B 0,C 180,E1 3322.243,E2 3322.243} C_VEL
LIN {X 0,Y 552.399,Z 529.66,A -85,B 0,C 180,E1 3326.867,E2 3326.867} C_VEL
LIN {X 0,Y 552.542,Z 529.66,A -85,B 0,C 180,E1 3331.564,E2 3331.564} C_VEL
LIN {X 0,Y 552.462,Z 529.66,A -85,B 0,C 180,E1 3336.272,E2 3336.272} C_VEL
LIN {X 0,Y 552.094,Z 529.66,A -85,B 0,C 180,E1 3342.629,E2 3342.629} C_VEL
LIN {X 0,Y 552.103,Z 529.66,A -85,B 0,C 180,E1 3347.496,E2 3347.496} C_VEL
LIN {X 0,Y 552.015,Z 529.66,A -85,B 0,C 180,E1 3352.501,E2 3352.501} C_VEL
LIN {X 0,Y 551.879,Z 529.66,A -85,B 0,C 180,E1 3357.698,E2 3357.698} C_VEL
LIN {X 0,Y 551.861,Z 529.66,A -85,B 0,C 180,E1 3363.152,E2 3363.152} C_VEL
LIN {X 0,Y 552.027,Z 529.66,A -85,B 0,C 180,E1 3368.954,E2 3368.954} C_VEL
LIN {X 0,Y 551.929,Z 529.66,A -85,B 0,C 180,E1 3375.303,E2 3375.303} C_VEL
LIN {X 0,Y 551.951,Z 529.66,A -85,B 0,C 180,E1 3381.036,E2 3381.036} C_VEL
LIN {X 0,Y 551.847,Z 529.66,A -85,B 0,C 180,E1 3386.844,E2 3386.844} C_VEL
LIN {X 0,Y 551.938,Z 529.66,A -85,B 0,C 180,E1 3392.302,E2 3392.302} C_VEL
LIN {X 0,Y 552.33,Z 529.768,A -85,B 0,C 180,E1 3396.325,E2 3396.325} C_VEL
LIN {X 0,Y 557.153,Z 546.512,A -85,B 0,C 180,E1 3396.772,E2 3396.772} C_VEL
LIN {X 0,Y 556.683,Z 582.7,A -85,B 0,C 180,E1 3397.527,E2 3397.527} C_VEL
LIN {X 0,Y 555.89,Z 617.3,A -85,B 0,C 180,E1 3398.918,E2 3398.918} C_VEL
LIN {X 0,Y 554.925,Z 648.712,A -85,B 0,C 180,E1 3400.867,E2 3400.867} C_VEL
LIN {X 0,Y 553.962,Z 677.195,A -85,B 0,C 180,E1 3403.378,E2 3403.378} C_VEL
LIN {X 0,Y 553.317,Z 700.36,A -85,B 0,C 180,E1 3406.192,E2 3406.192} C_VEL
LIN {X 0,Y 552.84,Z 719.686,A -85,B 0,C 180,E1 3409.474,E2 3409.474} C_VEL
LIN {X 0,Y 552.656,Z 733.411,A -85,B 0,C 180,E1 3412.94,E2 3412.94} C_VEL
LIN {X 0,Y 552.615,Z 740.804,A -85,B 0,C 180,E1 3416.084,E2 3416.084} C_VEL
LIN {X 0,Y 552.514,Z 743.472,A -85,B 0,C 180,E1 3418.433,E2 3418.433} C_VEL
LIN {X 0,Y 552.63,Z 743.417,A -85,B 0,C 180,E1 3421.563,E2 3421.563} C_VEL
LIN {X 0,Y 552.603,Z 739.19,A -85,B 0,C 180,E1 3424.697,E2 3424.697} C_VEL
LIN {X 0,Y 552.731,Z 729.091,A -85,B 0,C 180,E1 3428.238,E2 3428.238} C_VEL
LIN {X 0,Y 553.014,Z 713.589,A -85,B 0,C 180,E1 3431.607,E2 3431.607} C_VEL
LIN {X 0,Y 553.565,Z 692.391,A -85,B 0,C 180,E1 3434.787,E2 3434.787} C_VEL
LIN {X 0,Y 554.24,Z 669.209,A -85,B 0,C 180,E1 3437.325,E2 3437.325} C_VEL
LIN {X 0,Y 550.878,Z 656.753,A -85,B 0,C 180,E1 3438.56,E2 3438.56} C_VEL
LIN {X 0,Y 547.59,Z 645.278,A -85,B 0,C 180,E1 3439.569,E2 3439.569} C_VEL
LIN {X 0,Y 547.597,Z 643.457,A -85,B 0,C 180,E1 3439.699,E2 3439.699} C_VEL
LIN {X 0,Y 548.695,Z 611.352,A -85,B 0,C 180,E1 3441.579,E2 3441.579} C_VEL
LIN {X 0,Y 549.524,Z 577.333,A -85,B 0,C 180,E1 3442.853,E2 3442.853} C_VEL
LIN {X 0,Y 549.19,Z 544.234,A -85,B 0,C 180,E1 3443.526,E2 3443.526} C_VEL
LIN {X 0,Y 544.197,Z 529.66,A -85,B 0,C 180,E1 3444.051,E2 3444.051} C_VEL
LIN {X 0,Y 544.007,Z 529.66,A -85,B 0,C 180,E1 3449.95,E2 3449.95} C_VEL
LIN {X 0,Y 543.948,Z 529.66,A -85,B 0,C 180,E1 3455.628,E2 3455.628} C_VEL
LIN {X 0,Y 543.928,Z 529.66,A -85,B 0,C 180,E1 3461.742,E2 3461.742} C_VEL
LIN {X 0,Y 544.053,Z 529.66,A -85,B 0,C 180,E1 3468.267,E2 3468.267} C_VEL
LIN {X 0,Y 544.035,Z 529.66,A -85,B 0,C 180,E1 3473.545,E2 3473.545} C_VEL
LIN {X 0,Y 543.993,Z 529.66,A -85,B 0,C 180,E1 3479.302,E2 3479.302} C_VEL
LIN {X 0,Y 544.051,Z 530.297,A -85,B 0,C 180,E1 3481.322,E2 3481.322} C_VEL
LIN {X 0,Y 551.822,Z 552.053,A -85,B 0,C 180,E1 3482.077,E2 3482.077} C_VEL
LIN {X 0,Y 551.364,Z 595.136,A -85,B 0,C 180,E1 3482.865,E2 3482.865} C_VEL
LIN {X 0,Y 550.329,Z 631.013,A -85,B 0,C 180,E1 3484.127,E2 3484.127} C_VEL
LIN {X 0,Y 549.006,Z 666.953,A -85,B 0,C 180,E1 3486.084,E2 3486.084} C_VEL
LIN {X 0,Y 547.599,Z 699.272,A -85,B 0,C 180,E1 3488.586,E2 3488.586} C_VEL
LIN {X 0,Y 546.415,Z 727.044,A -85,B 0,C 180,E1 3491.484,E2 3491.484} C_VEL
LIN {X 0,Y 545.464,Z 751.937,A -85,B 0,C 180,E1 3494.99,E2 3494.99} C_VEL
LIN {X 0,Y 544.947,Z 769.653,A -85,B 0,C 180,E1 3498.419,E2 3498.419} C_VEL
LIN {X 0,Y 544.709,Z 782.685,A -85,B 0,C 180,E1 3502.039,E2 3502.039} C_VEL
LIN {X 0,Y 544.648,Z 790.9,A -85,B 0,C 180,E1 3505.835,E2 3505.835} C_VEL
LIN {X 0,Y 544.556,Z 794,A -85,B 0,C 180,E1 3510.001,E2 3510.001} C_VEL
LIN {X 0,Y 544.725,Z 792.179,A -85,B 0,C 180,E1 3513.177,E2 3513.177} C_VEL
LIN {X 0,Y 544.759,Z 784.898,A -85,B 0,C 180,E1 3517.161,E2 3517.161} C_VEL
LIN {X 0,Y 545.004,Z 771.381,A -85,B 0,C 180,E1 3521.176,E2 3521.176} C_VEL
LIN {X 0,Y 545.5,Z 753.016,A -85,B 0,C 180,E1 3524.826,E2 3524.826} C_VEL
LIN {X 0,Y 546.396,Z 728.776,A -85,B 0,C 180,E1 3528.31,E2 3528.31} C_VEL
LIN {X 0,Y 547.563,Z 700.404,A -85,B 0,C 180,E1 3531.311,E2 3531.311} C_VEL
LIN {X 0,Y 548.899,Z 668.466,A -85,B 0,C 180,E1 3533.815,E2 3533.815} C_VEL
LIN {X 0,Y 550.245,Z 632.666,A -85,B 0,C 180,E1 3535.803,E2 3535.803} C_VEL
LIN {X 0,Y 551.294,Z 595.677,A -85,B 0,C 180,E1 3537.123,E2 3537.123} C_VEL
LIN {X 0,Y 551.797,Z 550.664,A -85,B 0,C 180,E1 3537.944,E2 3537.944} C_VEL
LIN {X 0,Y 544.029,Z 529.66,A -85,B 0,C 180,E1 3538.741,E2 3538.741} C_VEL
LIN {X 0,Y 543.963,Z 529.66,A -85,B 0,C 180,E1 3543.699,E2 3543.699} C_VEL
LIN {X 0,Y 544.071,Z 529.66,A -85,B 0,C 180,E1 3549.637,E2 3549.637} C_VEL
LIN {X 0,Y 544.008,Z 529.66,A -85,B 0,C 180,E1 3556.155,E2 3556.155} C_VEL
LIN {X 0,Y 544.082,Z 529.66,A -85,B 0,C 180,E1 3562.402,E2 3562.402} C_VEL
LIN {X 0,Y 544.029,Z 529.66,A -85,B 0,C 180,E1 3568.199,E2 3568.199} C_VEL
LIN {X 0,Y 544.098,Z 529.66,A -85,B 0,C 180,E1 3573.66,E2 3573.66} C_VEL
LIN {X 0,Y 544.189,Z 529.66,A -85,B 0,C 180,E1 3578.873,E2 3578.873} C_VEL
LIN {X 0,Y 544.221,Z 529.66,A -85,B 0,C 180,E1 3583.905,E2 3583.905} C_VEL
LIN {X 0,Y 544.28,Z 529.66,A -85,B 0,C 180,E1 3590.427,E2 3590.427} C_VEL
LIN {X 0,Y 544.366,Z 529.66,A -85,B 0,C 180,E1 3595.232,E2 3595.232} C_VEL
LIN {X 0,Y 544.434,Z 529.66,A -85,B 0,C 180,E1 3600.002,E2 3600.002} C_VEL
LIN {X 0,Y 544.422,Z 529.66,A -85,B 0,C 180,E1 3604.772,E2 3604.772} C_VEL
LIN {X 0,Y 544.338,Z 529.66,A -85,B 0,C 180,E1 3609.576,E2 3609.576} C_VEL
LIN {X 0,Y 544.315,Z 529.66,A -85,B 0,C 180,E1 3614.45,E2 3614.45} C_VEL
LIN {X 0,Y 544.219,Z 529.66,A -85,B 0,C 180,E1 3619.481,E2 3619.481} C_VEL
LIN {X 0,Y 544.083,Z 529.66,A -85,B 0,C 180,E1 3624.585,E2 3624.585} C_VEL
LIN {X 0,Y 543.98,Z 529.66,A -85,B 0,C 180,E1 3630.689,E2 3630.689} C_VEL
LIN {X 0,Y 543.905,Z 529.66,A -85,B 0,C 180,E1 3636.431,E2 3636.431} C_VEL
LIN {X 0,Y 543.93,Z 529.66,A -85,B 0,C 180,E1 3641.747,E2 3641.747} C_VEL
LIN {X 0,Y 544.252,Z 529.66,A -85,B 0,C 180,E1 3647.418,E2 3647.418} C_VEL
LIN {X 0,Y 547.423,Z 547.352,A -85,B 0,C 180,E1 3647.772,E2 3647.772} C_VEL
LIN {X 0,Y 547.183,Z 624.24,A -85,B 0,C 180,E1 3648.899,E2 3648.899} C_VEL
LIN {X 0,Y 546.688,Z 652.118,A -85,B 0,C 180,E1 3649.914,E2 3649.914} C_VEL
LIN {X 0,Y 546.056,Z 677.975,A -85,B 0,C 180,E1 3651.491,E2 3651.491} C_VEL
LIN {X 0,Y 545.482,Z 701.139,A -85,B 0,C 180,E1 3653.621,E2 3653.621} C_VEL
LIN {X 0,Y 545.047,Z 719.755,A -85,B 0,C 180,E1 3656.16,E2 3656.16} C_VEL
LIN {X 0,Y 544.879,Z 732.368,A -85,B 0,C 180,E1 3658.744,E2 3658.744} C_VEL
LIN {X 0,Y 544.707,Z 741.249,A -85,B 0,C 180,E1 3661.903,E2 3661.903} C_VEL
LIN {X 0,Y 544.583,Z 743.503,A -85,B 0,C 180,E1 3663.682,E2 3663.682} C_VEL
LIN {X 0,Y 544.557,Z 743.568,A -85,B 0,C 180,E1 3666.13,E2 3666.13} C_VEL
LIN {X 0,Y 544.76,Z 738.477,A -85,B 0,C 180,E1 3669.279,E2 3669.279} C_VEL
LIN {X 0,Y 544.915,Z 727.662,A -85,B 0,C 180,E1 3672.264,E2 3672.264} C_VEL
LIN {X 0,Y 545.213,Z 711.788,A -85,B 0,C 180,E1 3674.961,E2 3674.961} C_VEL
LIN {X 0,Y 545.726,Z 691.072,A -85,B 0,C 180,E1 3677.321,E2 3677.321} C_VEL
LIN {X 0,Y 546.427,Z 665.649,A -85,B 0,C 180,E1 3679.256,E2 3679.256} C_VEL
LIN {X 0,Y 546.966,Z 638.484,A -85,B 0,C 180,E1 3680.571,E2 3680.571} C_VEL
LIN {X 0,Y 547.309,Z 611.309,A -85,B 0,C 180,E1 3681.277,E2 3681.277} C_VEL
LIN {X 0,Y 546.579,Z 539.247,A -85,B 0,C 180,E1 3682.274,E2 3682.274} C_VEL
LIN {X 0,Y 544.128,Z 529.66,A -85,B 0,C 180,E1 3682.534,E2 3682.534} C_VEL
LIN {X 0,Y 544.313,Z 529.66,A -85,B 0,C 180,E1 3688.411,E2 3688.411} C_VEL
LIN {X 0,Y 544.36,Z 529.66,A -85,B 0,C 180,E1 3693.177,E2 3693.177} C_VEL
LIN {X 0,Y 544.249,Z 529.66,A -85,B 0,C 180,E1 3697.968,E2 3697.968} C_VEL
LIN {X 0,Y 544.173,Z 529.66,A -85,B 0,C 180,E1 3702.816,E2 3702.816} C_VEL
LIN {X 0,Y 544.173,Z 529.66,A -85,B 0,C 180,E1 3707.759,E2 3707.759} C_VEL
LIN {X 0,Y 544.071,Z 529.66,A -85,B 0,C 180,E1 3712.848,E2 3712.848} C_VEL
LIN {X 0,Y 543.959,Z 529.66,A -85,B 0,C 180,E1 3718.137,E2 3718.137} C_VEL
LIN {X 0,Y 543.958,Z 529.66,A -85,B 0,C 180,E1 3723.697,E2 3723.697} C_VEL
LIN {X 0,Y 544.129,Z 529.66,A -85,B 0,C 180,E1 3729.056,E2 3729.056} C_VEL
LIN {X 0,Y 543.955,Z 529.66,A -85,B 0,C 180,E1 3733.909,E2 3733.909} C_VEL
LIN {X 0,Y 544.064,Z 529.66,A -85,B 0,C 180,E1 3738.491,E2 3738.491} C_VEL
LIN {X 0,Y 543.957,Z 529.66,A -85,B 0,C 180,E1 3744.367,E2 3744.367} C_VEL
LIN {X 0,Y 543.973,Z 529.66,A -85,B 0,C 180,E1 3750.043,E2 3750.043} C_VEL
LIN {X 0,Y 544.341,Z 529.66,A -85,B 0,C 180,E1 3755.953,E2 3755.953} C_VEL
LIN {X 0,Y 549.886,Z 547.896,A -85,B 0,C 180,E1 3756.467,E2 3756.467} C_VEL
LIN {X 0,Y 549.334,Z 583.944,A -85,B 0,C 180,E1 3757.25,E2 3757.25} C_VEL
LIN {X 0,Y 548.469,Z 617.287,A -85,B 0,C 180,E1 3758.618,E2 3758.618} C_VEL
LIN {X 0,Y 547.373,Z 648.801,A -85,B 0,C 180,E1 3760.6,E2 3760.6} C_VEL
LIN {X 0,Y 546.283,Z 677.186,A -85,B 0,C 180,E1 3763.138,E2 3763.138} C_VEL
LIN {X 0,Y 545.555,Z 700.351,A -85,B 0,C 180,E1 3765.992,E2 3765.992} C_VEL
LIN {X 0,Y 545.006,Z 719.685,A -85,B 0,C 180,E1 3769.321,E2 3769.321} C_VEL
LIN {X 0,Y 544.768,Z 733.41,A -85,B 0,C 180,E1 3772.837,E2 3772.837} C_VEL
LIN {X 0,Y 544.697,Z 740.398,A -85,B 0,C 180,E1 3775.794,E2 3775.794} C_VEL
LIN {X 0,Y 544.613,Z 743.473,A -85,B 0,C 180,E1 3778.41,E2 3778.41} C_VEL
LIN {X 0,Y 544.727,Z 743.419,A -85,B 0,C 180,E1 3781.585,E2 3781.585} C_VEL
LIN {X 0,Y 544.713,Z 739.194,A -85,B 0,C 180,E1 3784.765,E2 3784.765} C_VEL
LIN {X 0,Y 544.854,Z 729.093,A -85,B 0,C 180,E1 3788.358,E2 3788.358} C_VEL
LIN {X 0,Y 545.153,Z 713.592,A -85,B 0,C 180,E1 3791.777,E2 3791.777} C_VEL
LIN {X 0,Y 545.807,Z 692.224,A -85,B 0,C 180,E1 3795.024,E2 3795.024} C_VEL
LIN {X 0,Y 546.686,Z 666.771,A -85,B 0,C 180,E1 3797.808,E2 3797.808} C_VEL
LIN {X 0,Y 547.597,Z 643.457,A -85,B 0,C 180,E1 3799.699,E2 3799.699} C_VEL
LIN {X 0,Y 544.445,Z 629.491,A -85,B 0,C 180,E1 3800.761,E2 3800.761} C_VEL
LIN {X 0,Y 541.177,Z 616.869,A -85,B 0,C 180,E1 3801.615,E2 3801.615} C_VEL
LIN {X 0,Y 541.151,Z 614.891,A -85,B 0,C 180,E1 3801.718,E2 3801.718} C_VEL
LIN {X 0,Y 542.082,Z 582.041,A -85,B 0,C 180,E1 3803.042,E2 3803.042} C_VEL
LIN {X 0,Y 542.157,Z 546.638,A -85,B 0,C 180,E1 3803.816,E2 3803.816} C_VEL
LIN {X 0,Y 536.243,Z 529.66,A -85,B 0,C 180,E1 3804.417,E2 3804.417} C_VEL
LIN {X 0,Y 536.098,Z 529.66,A -85,B 0,C 180,E1 3810.439,E2 3810.439} C_VEL
LIN {X 0,Y 536.023,Z 529.66,A -85,B 0,C 180,E1 3816.238,E2 3816.238} C_VEL
LIN {X 0,Y 535.941,Z 529.66,A -85,B 0,C 180,E1 3822.508,E2 3822.508} C_VEL
LIN {X 0,Y 536.048,Z 529.66,A -85,B 0,C 180,E1 3827.5,E2 3827.5} C_VEL
LIN {X 0,Y 536.117,Z 529.66,A -85,B 0,C 180,E1 3833.767,E2 3833.767} C_VEL
LIN {X 0,Y 536.081,Z 529.66,A -85,B 0,C 180,E1 3839.558,E2 3839.558} C_VEL
LIN {X 0,Y 536.134,Z 529.66,A -85,B 0,C 180,E1 3840.835,E2 3840.835} C_VEL
LIN {X 0,Y 544.839,Z 553.911,A -85,B 0,C 180,E1 3841.714,E2 3841.714} C_VEL
LIN {X 0,Y 544.297,Z 596.146,A -85,B 0,C 180,E1 3842.512,E2 3842.512} C_VEL
LIN {X 0,Y 543.137,Z 631.751,A -85,B 0,C 180,E1 3843.792,E2 3843.792} C_VEL
LIN {X 0,Y 541.68,Z 666.949,A -85,B 0,C 180,E1 3845.739,E2 3845.739} C_VEL
LIN {X 0,Y 540.124,Z 699.337,A -85,B 0,C 180,E1 3848.281,E2 3848.281} C_VEL
LIN {X 0,Y 538.764,Z 727.044,A -85,B 0,C 180,E1 3851.211,E2 3851.211} C_VEL
LIN {X 0,Y 537.686,Z 751.814,A -85,B 0,C 180,E1 3854.746,E2 3854.746} C_VEL
LIN {X 0,Y 537.1,Z 769.654,A -85,B 0,C 180,E1 3858.248,E2 3858.248} C_VEL
LIN {X 0,Y 536.84,Z 782.685,A -85,B 0,C 180,E1 3861.921,E2 3861.921} C_VEL
LIN {X 0,Y 536.746,Z 790.9,A -85,B 0,C 180,E1 3865.773,E2 3865.773} C_VEL
LIN {X 0,Y 536.682,Z 794,A -85,B 0,C 180,E1 3870.001,E2 3870.001} C_VEL
LIN {X 0,Y 536.807,Z 791.215,A -85,B 0,C 180,E1 3874.014,E2 3874.014} C_VEL
LIN {X 0,Y 536.885,Z 782.679,A -85,B 0,C 180,E1 3878.079,E2 3878.079} C_VEL
LIN {X 0,Y 537.109,Z 769.648,A -85,B 0,C 180,E1 3881.753,E2 3881.753} C_VEL
LIN {X 0,Y 537.759,Z 750.598,A -85,B 0,C 180,E1 3885.461,E2 3885.461} C_VEL
LIN {X 0,Y 538.766,Z 727.032,A -85,B 0,C 180,E1 3888.79,E2 3888.79} C_VEL
LIN {X 0,Y 540.171,Z 698.232,A -85,B 0,C 180,E1 3891.821,E2 3891.821} C_VEL
LIN {X 0,Y 541.74,Z 665.304,A -85,B 0,C 180,E1 3894.369,E2 3894.369} C_VEL
LIN {X 0,Y 543.208,Z 630.411,A -85,B 0,C 180,E1 3896.266,E2 3896.266} C_VEL
LIN {X 0,Y 544.335,Z 593.993,A -85,B 0,C 180,E1 3897.547,E2 3897.547} C_VEL
LIN {X 0,Y 544.486,Z 551.483,A -85,B 0,C 180,E1 3898.341,E2 3898.341} C_VEL
LIN {X 0,Y 536.14,Z 529.66,A -85,B 0,C 180,E1 3899.187,E2 3899.187} C_VEL
LIN {X 0,Y 536.064,Z 529.66,A -85,B 0,C 180,E1 3905.285,E2 3905.285} C_VEL
LIN {X 0,Y 536.059,Z 529.66,A -85,B 0,C 180,E1 3910.536,E2 3910.536} C_VEL
LIN {X 0,Y 536.036,Z 529.66,A -85,B 0,C 180,E1 3917.049,E2 3917.049} C_VEL
LIN {X 0,Y 536.15,Z 529.66,A -85,B 0,C 180,E1 3922.006,E2 3922.006} C_VEL
LIN {X 0,Y 536.072,Z 529.66,A -85,B 0,C 180,E1 3927.671,E2 3927.671} C_VEL
LIN {X 0,Y 536.164,Z 529.66,A -85,B 0,C 180,E1 3933.239,E2 3933.239} C_VEL
LIN {X 0,Y 536.229,Z 529.66,A -85,B 0,C 180,E1 3938.544,E2 3938.544} C_VEL
LIN {X 0,Y 536.308,Z 529.66,A -85,B 0,C 180,E1 3943.661,E2 3943.661} C_VEL
LIN {X 0,Y 536.361,Z 529.66,A -85,B 0,C 180,E1 3950.284,E2 3950.284} C_VEL
LIN {X 0,Y 536.465,Z 529.66,A -85,B 0,C 180,E1 3955.162,E2 3955.162} C_VEL
LIN {X 0,Y 536.541,Z 529.66,A -85,B 0,C 180,E1 3960.002,E2 3960.002} C_VEL
LIN {X 0,Y 536.508,Z 529.66,A -85,B 0,C 180,E1 3964.842,E2 3964.842} C_VEL
LIN {X 0,Y 536.369,Z 529.66,A -85,B 0,C 180,E1 3970.041,E2 3970.041} C_VEL
LIN {X 0,Y 536.375,Z 529.66,A -85,B 0,C 180,E1 3974.669,E2 3974.669} C_VEL
LIN {X 0,Y 536.307,Z 529.66,A -85,B 0,C 180,E1 3979.735,E2 3979.735} C_VEL
LIN {X 0,Y 536.076,Z 529.66,A -85,B 0,C 180,E1 3985.74,E2 3985.74} C_VEL
LIN {X 0,Y 536.076,Z 529.66,A -85,B 0,C 180,E1 3990.445,E2 3990.445} C_VEL
